  // No operation or process is active
  CmdMessageState.EMPTY               :;
  // Created but not yet started
  CmdMessageState.CREATED             :;
  // Buffered and awaiting execution
  CmdMessageState.BUFFERED            : CommandBuffered    := TRUE;
                                        ParameterAccepted  := TRUE;
  // Buffered in planner for future execution
  CmdMessageState.BUFFERED_IN_PLANNER : CommandBuffered    := TRUE;
                                        ParameterAccepted  := TRUE;
  // Currently active and in progress
  CmdMessageState.ACTIVE              :;
  // Interrupted and awaiting continuation
  CmdMessageState.INTERRUPTED         :;  
  // Requested for abort
  CmdMessageState.ABORT_REQUEST       :;
  // Successfully completed
  CmdMessageState.DONE                : Done               := TRUE;
                                        Busy               := FALSE;
  // Aborted before completion
  CmdMessageState.ABORTED             : Busy               := FALSE;
  // Encountered an error during execution
  CmdMessageState.ERROR               : Error              := TRUE;
                                        Busy               := FALSE;
END_CASE
                
END_METHOD

METHOD INTERNAL ParseResponsePayload : DINT
VAR_INPUT
  /// Response data
  ResponseData : RobotLibraryResponseDataFB;
  /// Timestamp
  Timestamp    : SystemTime;  
END_VAR
VAR
  /// Parameter count
 _parameterCnt : DINT;
END_VAR
// Table 6-445: Received CMD payload (RC to PLC) of "RedefineTrackingPos"
// --------------------------
// Header
// --------------------------
// Byte 00 : USINT      - ParSeq | State     
// Byte 01 : SINT       - AlarmMessageSeverity    
// Byte 02 : UINT       - AlarmMessageCode HB
// Byte 03 :            - AlarmMessageCode LB
// --------------------------
// Datablock
// --------------------------
// Byte 04 : USINT InvocationCounter;
// Byte 05 : SINT  Reserved;
// Byte 06 : INT   OriginID;
// Byte 07 :       OriginID;
                  // call base implementation to parse the header from payload buffer
ResponseData.PayloadPtr := SUPER^.ParseResponsePayload(ResponseData := ResponseData, Timestamp := Timestamp);

// copy parsed header to response
_response.ParSeq                := _rspHeader.ParSeq;
_response.State                 := _rspHeader.State;
_response.AlarmMessageSeverity  := _rspHeader.AlarmMessageSeverity;
_response.AlarmMessageCode      := _rspHeader.AlarmMessageCode;

// Check payload remaining ? 
IF ( ResponseData.IsPayloadRemaining)
THEN 
  // Get Response.InvocationCounter
 _response.InvocationCounter := ResponseData.GetUsint();
  // inc parameter counter
 _parameterCnt := _parameterCnt + 1;
END_IF


// Check payload remaining ? 
IF ( ResponseData.IsPayloadRemaining)
THEN 
  // Get Response.Reserved
  _response.Reserved := ResponseData.GetSint();
  // inc parameter counter
 _parameterCnt := _parameterCnt + 1;
END_IF


// Check payload remaining ? 
IF ( ResponseData.IsPayloadRemaining)
THEN 
  // Get Response.InvocationCounter
 _response.OriginID := ResponseData.GetInt();
  // inc parameter counter
 _parameterCnt := _parameterCnt + 1;
END_IF

 
// Create logging
ParseResponsePayloadLog(ResponseData := ResponseData, Timestamp := Timestamp, ParameterCnt := _parameterCnt);
                
END_METHOD

METHOD INTERNAL ParseResponsePayloadLog
VAR_INPUT
  /// Response data
  ResponseData : RobotLibraryResponseDataFB;
  /// Timestamp
  Timestamp    : SystemTime;  
  /// Parameter count
  ParameterCnt : DINT;
END_VAR
                  // Create log entry for Parameter start
CreateLogMessagePara1 ( Timestamp   := Timestamp,
                        MessageType := MessageType.CMD,
                        Severity    := Severity.DEBUG,
                        MessageCode := 0,
                        MessageText := '{1} parameter(s) to parse from the response data:',
                        Para1       := DINT_TO_STRING(ParameterCnt));
                        

// Return if no parameter is remaining...
IF ( ParameterCnt = 0 ) THEN RETURN; END_IF
// dec remaining parameter(s)                        
ParameterCnt := ParameterCnt - 1;
// Create log entry for InvocationCounter
CreateLogMessagePara1 ( Timestamp   := Timestamp,
                        MessageType := MessageType.CMD,
                        Severity    := Severity.DEBUG,
                        MessageCode := 0,
                        MessageText := 'Response.InvocationCounter = {1}',
                        Para1       :=  USINT_TO_STRING(_response.InvocationCounter));


// Return if no parameter is remaining...
IF ( ParameterCnt = 0 ) THEN RETURN; END_IF
// dec remaining parameter(s)                        
ParameterCnt := ParameterCnt - 1;
// Create log entry for Reserve
CreateLogMessagePara1 ( Timestamp   := Timestamp,
                        MessageType := MessageType.CMD,
                        Severity    := Severity.DEBUG,
                        MessageCode := 0,
                        MessageText := 'Response.Reserve = {1}',
                        Para1       :=  SINT_TO_STRING(_response.Reserved));


// Return if no parameter is remaining...
IF ( ParameterCnt = 0 ) THEN RETURN; END_IF
// dec remaining parameter(s)                        
ParameterCnt := ParameterCnt - 1;
// Create log entry for OriginID
CreateLogMessagePara1 ( Timestamp   := Timestamp,
                        MessageType := MessageType.CMD,
                        Severity    := Severity.DEBUG,
                        MessageCode := 0,
                        MessageText := 'Response.OriginID = {1}',
                        Para1       :=  INT_TO_STRING(_response.OriginID));
                
END_METHOD

METHOD PROTECTED Reset : DINT
VAR_INPUT
END_VAR
                  Reset := SUPER^.Reset();

Done               := FALSE;
Busy               := FALSE;
CommandBuffered    := FALSE;
ParameterAccepted  := FALSE;

                
END_METHOD
END_FUNCTION_BLOCK

/// Synchronize robot with conveyor
FUNCTION_BLOCK MC_SyncToConveyorFB EXTENDS RobotLibraryBaseEnableFB
// ------------------------------------------------------------------------- 
//  SRCI Robot Library                                                
// ------------------------------------------------------------------------- 
//                                                                           
//  Object:      SyncToConveyorFB                                       
//  Author:      Thorsten Brach                                                
//  Date:        2024-06-11
//
//  Description:                                              
//   
//                                                                           
//  Copyright: 
//    (C) 2024 Thorsten Brach. All rights reserved                                                                                                                                            
//             Licensed under the MIT License.
//                                                                           
//  Disclaimer:                                                                           
//    This project is provided without any guarantee and can be used for   
//    private and commercial purposes. Any use is at the user’s 
//    own risk and responsibility.
//
// -------------------------------------------------------------------------
VAR_INPUT
  /// Command parameter 
  ParCmd            : SyncToConveyorParCmd;      
END_VAR

VAR_OUTPUT
  /// Command is transferred and confirmed by the RC
  CommandBuffered   : BOOL;
  /// The command takes control of the motion of the according axis group
  Active            : BOOL;
  /// The command was aborted by another command.
  CommandAborted    : BOOL;
  /// Receiving of input parameter values has been acknowledged by RC
  ParameterAccepted : BOOL;
  /// Command output 
  OutCmd            : SyncToConveyorOutCmd;      
END_VAR

VAR
  /// internal copy of command parameter 
 _parCmd            : SyncToConveyorParCmd;
  /// command data to send
 _command           : SyncToConveyorSendData;
  /// response data received
 _response          : SyncToConveyorRecvData;      
END_VAR

            SUPER^(AxesGroup := AxesGroup);
          

METHOD INTERNAL CheckAddParameter : BOOL
VAR_INPUT
  /// Payload pointer
  PayloadPtr : UDINT;
END_VAR
VAR
  /// Payload as byte array
  Payload    : ARRAY [1..SIZEOF(_command)] OF BYTE;
  /// Null Byte array 
  Null       : ARRAY [1..SIZEOF(_command)] OF BYTE;
  /// Data length to compare
  DataLen    : UDINT;
END_VAR
                  // Payload pointer must be decreased by one byte, because ADR(Payload) is already one byte !
PayloadPtr := LIMIT (0, PayloadPtr - 1, SIZEOF(Payload) -1);
// Convert command struct to payload array
SysDepMemCpy( pDest := ADR(Payload), pSrc := ADR(_command), DataLen := SIZEOF(_command));
// Calculate the data length to compare - at least one byte must be compared !
DataLen := LIMIT(1, SIZEOF(Payload) - PayloadPtr, SIZEOF(Payload)); 
// Compare Payload-Array with Null-Byte-Array
CheckAddParameter := SysDepMemCmp( pData1 := ADR(Payload) + PayloadPtr , pData2 := ADR(Null), DataLen := DataLen) <>  RobotLibraryConstants.OK ;
                
END_METHOD

METHOD PROTECTED CheckFunctionSupported : BOOL
VAR_IN_OUT
  /// Robot assignment of function
  AxesGroup : AxesGroup; 
END_VAR
                  CheckFunctionSupported := AxesGroup.State.RobotData.RCSupportedFunctions.SyncToConveyor;

IF ( NOT CheckFunctionSupported )
THEN
  // call base implementation for set error and create log entry
  SUPER^.CheckFunctionSupported(AxesGroup := AxesGroup);
END_IF
                
END_METHOD

METHOD PROTECTED CheckParameterChanged : BOOL
VAR_IN_OUT
  /// Robot assignment of function
  AxesGroup    : AxesGroup; 
END_VAR
                  // Check ParCmd Size is > 0, because MemCmp does not work correctly with size = 0
IF (SIZEOF(ParCmd) = 0) OR (_stepCmd = 0)
THEN 
  RETURN;
END_IF

// compare memory 
_parameterChanged := ( SysDepMemCmp(pData1 := ADR(ParCmd), pData2 := ADR(_parCmd), DataLen := SIZEOF(ParCmd)) <> RobotLibraryConstants.OK );

// check parameter valid ?
_parameterValid   := CheckParameterValid( AxesGroup := AxesGroup );

IF ((  _parameterChanged        )  AND 
    (  _parameterValid          )) OR
    (  _parameterUpdateInternal )  
THEN  
  // Create log entry for parameter changed event
  CreateLogMessagePara1 ( Timestamp   := AxesGroup.State.SystemTime,
                          MessageType := MessageType.CMD,
                          Severity    := Severity.DEBUG,
                          MessageCode := 0,
                          MessageText := 'NotifyParameterChanged Event {1}',
                          Para1       :=  '' );

  // reset internal flag for send parameter update
 _parameterUpdateInternal := FALSE;
  // update internal copy of parameters 
 _parCmd := ParCmd;
  // inc parameter sequence
 _command.ParSeq := _command.ParSeq + 1;
  // update command data  
  CommandData := CreateCommandPayload(AxesGroup := AxesGroup); // ( Access via reference to rCommandFB in ACR )
  // notify active command register 
  AxesGroup.Acyclic.ActiveCommandRegister.NotifyParameterChanged := _uniqueID;
  // Reset parameter accepted flag
  ParameterAccepted := FALSE;  
END_IF
                
END_METHOD

METHOD PROTECTED CheckParameterValid : BOOL
VAR_IN_OUT
  /// Robot assignment of function
  AxesGroup : AxesGroup; 
END_VAR
                  CheckParameterValid := TRUE;


// Check ParCmd.ConveyorNo valid ? 
IF (( ParCmd.ConveyorNo <   0 ) OR  
    ( ParCmd.ConveyorNo > 255 ))
THEN
  // Parameter not valid
  CheckParameterValid := FALSE;
  // Set error
  SetError( ErrorID := RobotLibraryErrorIdEnum.ERR_INVALID_PAR_CMD, Overwrite := TRUE );
  // Create log entry
  CreateLogMessagePara1 ( Timestamp   := AxesGroup.State.SystemTime,
                          MessageType := MessageType.CMD,
                          Severity    := Severity.ERROR,
                          MessageCode := ErrorID,
                          MessageText := 'Invalid Parameter ParCmd.ConveyorNo = {1}',
                          Para1       :=  USINT_TO_STRING(ParCmd.ConveyorNo));
  RETURN;                          
END_IF


// Check ParCmd.FrameNo valid ? 
IF (( ParCmd.FrameNo <   0                                                 ) OR  
    ( ParCmd.FrameNo > 254                                                 ) OR
    ( ParCmd.FrameNo > AxesGroup.State.ConfigurationData.HighestFrameIndex ) OR
    ( ParCmd.FrameNo > AxesGroup.State.UnifiedFrameIndex                   ))         
THEN
  // Parameter not valid
  CheckParameterValid := FALSE;
  
  // Check FrameNo available on RC ? 
  IF ( ParCmd.FrameNo > AxesGroup.State.ConfigurationData.HighestFrameIndex )
  THEN
    SetError( ErrorID := RobotLibraryErrorIdEnum.ERR_FRAMENO_UNAVAILABLE, Overwrite := TRUE );
  ELSE
    SetError( ErrorID := RobotLibraryErrorIdEnum.ERR_FRAMENO_RANGE, Overwrite := TRUE );
	END_IF  
  
  // Create log entry
  CreateLogMessagePara1 ( Timestamp   := AxesGroup.State.SystemTime,
                          MessageType := MessageType.CMD,
                          Severity    := Severity.ERROR,
                          MessageCode := ErrorID,
                          MessageText := 'Invalid Parameter ParCmd.FrameNo = {1}',
                          Para1       :=  USINT_TO_STRING(ParCmd.FrameNo));
  RETURN;                          
END_IF


// Check ParCmd.SyncInMode valid ? 
IF (( ParCmd.SyncInMode <> SyncInMode.IN_SYNC_IN_ZONE ) AND  
    ( ParCmd.SyncInMode <> SyncInMode.AFTER_DISTANCE  ) AND
    ( ParCmd.SyncInMode <> SyncInMode.AFTER_TIME      ) AND
    ( ParCmd.SyncInMode <> SyncInMode.IMMEDIATELY     ))
THEN
  // Parameter not valid
  CheckParameterValid := FALSE;
  // Set error
  SetError( ErrorID := RobotLibraryErrorIdEnum.ERR_INVALID_PAR_CMD, Overwrite := TRUE );
  // Create log entry
  CreateLogMessagePara1 ( Timestamp   := AxesGroup.State.SystemTime,
                          MessageType := MessageType.CMD,
                          Severity    := Severity.ERROR,
                          MessageCode := ErrorID,
                          MessageText := 'Invalid Parameter ParCmd.SyncInMode = {1}',
                          Para1       :=  SYNC_IN_MODE_TO_STRING(ParCmd.SyncInMode));
  RETURN;                          
END_IF


// Check ParCmd.SyncInParameter valid ? 
IF ( SysDepIsValidReal(ParCmd.SyncInParameter) = FALSE ) 
THEN
  // Parameter not valid
  CheckParameterValid := FALSE;
  // Set error
  SetError( ErrorID := RobotLibraryErrorIdEnum.ERR_INVALID_PAR_CMD, Overwrite := TRUE );
  
  // Create log entry
  CreateLogMessagePara1 ( Timestamp   := AxesGroup.State.SystemTime,
                          MessageType := MessageType.CMD,
                          Severity    := Severity.ERROR,
                          MessageCode := ErrorID,
                          MessageText := 'Invalid Parameter ParCmd.SyncInParameter = {1}',
                          Para1       := VALID_REAL_TO_STRING(ParCmd.SyncInParameter));
  RETURN;                          
END_IF


// Check ParCmd.MaxVelocity valid ? 
IF ( SysDepIsValidReal(ParCmd.MaxVelocity) = FALSE ) 
THEN
  // Parameter not valid
  CheckParameterValid := FALSE;
  // Set error
  SetError( ErrorID := RobotLibraryErrorIdEnum.ERR_INVALID_PAR_CMD, Overwrite := TRUE );
  
  // Create log entry
  CreateLogMessagePara1 ( Timestamp   := AxesGroup.State.SystemTime,
                          MessageType := MessageType.CMD,
                          Severity    := Severity.ERROR,
                          MessageCode := ErrorID,
                          MessageText := 'Invalid Parameter ParCmd.MaxVelocity = {1}',
                          Para1       := VALID_REAL_TO_STRING(ParCmd.MaxVelocity));
  RETURN;                          
END_IF


// Check ParCmd.MaxAcceleration valid ? 
IF ( SysDepIsValidReal(ParCmd.MaxAcceleration) = FALSE ) 
THEN
  // Parameter not valid
  CheckParameterValid := FALSE;
  // Set error
  SetError( ErrorID := RobotLibraryErrorIdEnum.ERR_INVALID_PAR_CMD, Overwrite := TRUE );
  
  // Create log entry
  CreateLogMessagePara1 ( Timestamp   := AxesGroup.State.SystemTime,
                          MessageType := MessageType.CMD,
                          Severity    := Severity.ERROR,
                          MessageCode := ErrorID,
                          MessageText := 'Invalid Parameter ParCmd.MaxAcceleration = {1}',
                          Para1       := VALID_REAL_TO_STRING(ParCmd.MaxAcceleration));
  RETURN;                          
END_IF


// Check ParCmd.ListenerID valid ? 
IF (( ParCmd.ListenerID <   0 ) OR  
    ( ParCmd.ListenerID > 127 ))
THEN
  // Parameter not valid
  CheckParameterValid := FALSE;
  // Set error
  SetError( ErrorID := RobotLibraryErrorIdEnum.ERR_INVALID_PAR_CMD, Overwrite := TRUE );
  // Create log entry
  CreateLogMessagePara1 ( Timestamp   := AxesGroup.State.SystemTime,
                          MessageType := MessageType.CMD,
                          Severity    := Severity.ERROR,
                          MessageCode := ErrorID,
                          MessageText := 'Invalid Parameter ParCmd.ListenerID = {1}',
                          Para1       :=  SINT_TO_STRING(ParCmd.ListenerID));
  RETURN;                          
END_IF
                
END_METHOD

METHOD INTERNAL CreateCommandPayload : RobotLibraryCommandDataFB
VAR_IN_OUT
  /// Robot assignment of function
  AxesGroup : AxesGroup; 
END_VAR
VAR
  /// internal index for loops
 _idx          : DINT;
  /// Parameter count
 _parameterCnt : DINT;
END_VAR
// Table 6-452: Sent CMD payload (PLC to RC) of "SyncToConveyor"
// --------------------------
// Header
// --------------------------
// Byte 00 : UINT       - Type HB     
// Byte 01 :            - Type LB    
// Byte 02 : USINT      - Reserve | ExecutionMode
// Byte 03 : USINT      - ParSeq  | Priority
// --------------------------
// Datablock
// --------------------------
// Byte 04 : SINT       - EmitterID[0]
// Byte 05 : SINT       - EmitterID[1]
// Byte 06 : SINT       - EmitterID[2]
// Byte 07 : SINT       - EmitterID[3]
// Byte 08 : SINT       - ListenerID
// Byte 09 : BYTE       - Reserved
// Byte 10 : USINT      - ConveyorNo
// Byte 11 : USINT      - FrameNo
// Byte 12 : USINT      - SyncInMode
// Byte 13 : REAL       - SyncInParameter HW HB
// Byte 14 :            - SyncInParameter HW LB
// Byte 15 :            - SyncInParameter LW HB
// Byte 16 :            - SyncInParameter LW LB
// Byte 17 : REAL       - MaxVelocity     HW HB
// Byte 18 :            - MaxVelocity     HW LB
// Byte 19 :            - MaxVelocity     LW HB
// Byte 20 :            - MaxVelocity     LW LB
// Byte 21 : REAL       - MaxAcceleration HW HB
// Byte 22 :            - MaxAcceleration HW LB
// Byte 23 :            - MaxAcceleration LW HB
// Byte 24 :            - MaxAcceleration LW LB
// --------------------------
                  // set command parameter 
_command.CmdTyp          :=  CmdType.SyncToConveyor;
_command.ExecMode        :=  ExecMode;
_command.ParSeq          := _command.ParSeq;
_command.Priority        :=  Priority;
_command.EmitterID[0]    := 0;
_command.EmitterID[1]    := 0;
_command.EmitterID[2]    := 0;
_command.EmitterID[3]    := 0;
_command.ListenerID      := _parCmd.ListenerID;
_command.Reserve         := 0;
_command.ConveyorNo      := _parCmd.ConveyorNo;
_command.FrameNo         := _parCmd.FrameNo;
_command.SyncInMode      := _parCmd.SyncInMode;
_command.SyncInParameter := _parCmd.SyncInParameter;
_command.MaxVelocity     := _parCmd.MaxVelocity;
_command.MaxAcceleration := _parCmd.MaxAcceleration;

// copy command data to header
_cmdHeader := _command;
// call base implementation to copy header to payload buffer
CreateCommandPayload := SUPER^.CreateCommandPayload(AxesGroup := AxesGroup);


FOR _idx := 0 TO 3 
DO
  // Check parameter must be added ? 
  IF ( CheckAddParameter(CreateCommandPayload.PayloadPtr))
  THEN
    // add command.EmitterID[x]
    CreateCommandPayload.AddSint(_command.EmitterID[_idx]);
    // inc parameter counter
   _parameterCnt := _parameterCnt + 1;  
  END_IF
END_FOR


// Check parameter must be added ? 
IF ( CheckAddParameter(CreateCommandPayload.PayloadPtr))
THEN
  // add command.ListenerID
  CreateCommandPayload.AddSint(_command.ListenerID);
  // inc parameter counter
 _parameterCnt := _parameterCnt + 1;  
END_IF


// Check parameter must be added ? 
IF ( CheckAddParameter(CreateCommandPayload.PayloadPtr))
THEN
  // add command.Reserve
  CreateCommandPayload.AddByte(_command.Reserve);
  // inc parameter counter
 _parameterCnt := _parameterCnt + 1;  
END_IF


// Check parameter must be added ? 
IF ( CheckAddParameter(CreateCommandPayload.PayloadPtr))
THEN
  // add command.ConveyorNo
  CreateCommandPayload.AddUsint(_command.ConveyorNo);
  // inc parameter counter
 _parameterCnt := _parameterCnt + 1;  
END_IF


// Check parameter must be added ? 
IF ( CheckAddParameter(CreateCommandPayload.PayloadPtr))
THEN
  // add command.FrameNo
  CreateCommandPayload.AddUsint(_command.FrameNo);
  // inc parameter counter
 _parameterCnt := _parameterCnt + 1;  
END_IF


// Check parameter must be added ? 
IF ( CheckAddParameter(CreateCommandPayload.PayloadPtr))
THEN
  // add command.SyncInMode
  CreateCommandPayload.AddUsint(_command.SyncInMode);
  // inc parameter counter
 _parameterCnt := _parameterCnt + 1;  
END_IF


// Check parameter must be added ? 
IF ( CheckAddParameter(CreateCommandPayload.PayloadPtr))
THEN
  // add command.SyncInParameter
  CreateCommandPayload.AddReal(_command.SyncInParameter);
  // inc parameter counter
 _parameterCnt := _parameterCnt + 1;  
END_IF


// Check parameter must be added ? 
IF ( CheckAddParameter(CreateCommandPayload.PayloadPtr))
THEN
  // add command.MaxVelocity
  CreateCommandPayload.AddReal(_command.MaxVelocity);
  // inc parameter counter
 _parameterCnt := _parameterCnt + 1;  
END_IF


// Check parameter must be added ? 
IF ( CheckAddParameter(CreateCommandPayload.PayloadPtr))
THEN
  // add command.MaxAcceleration
  CreateCommandPayload.AddReal(_command.MaxAcceleration);
  // inc parameter counter
 _parameterCnt := _parameterCnt + 1;  
END_IF
  
 
// Create logging
CreateCommandPayloadLog(AxesGroup := AxesGroup, ParameterCnt := _parameterCnt);
                
END_METHOD

METHOD INTERNAL CreateCommandPayloadLog 
VAR_IN_OUT
  /// Robot assignment of function
  AxesGroup : AxesGroup; 
END_VAR
VAR_INPUT
  /// Parameter count
  ParameterCnt : DINT;
END_VAR
VAR 
  /// internal index for loops
 _idx : DINT;
END_VAR
                  // Create log entry for Parameter start
CreateLogMessagePara1 ( Timestamp   := AxesGroup.State.SystemTime,
                        MessageType := MessageType.CMD,
                        Severity    := Severity.DEBUG,
                        MessageCode := 0,
                        MessageText := 'Create command payload with {1} parameter(s) :',
                        Para1       := DINT_TO_STRING(ParameterCnt));

// Create log entry for EmitterID[x]
FOR _idx := 0 TO 3
DO
  // Return if no parameter is remaining...
  IF ( ParameterCnt = 0 ) THEN RETURN; END_IF
  // dec remaining parameter(s)                        
  ParameterCnt := ParameterCnt - 1;
  // Create log entry for Command.EmitterID
  CreateLogMessagePara2 ( Timestamp   := AxesGroup.State.SystemTime,
                          MessageType := MessageType.CMD,
                          Severity    := Severity.DEBUG,
                          MessageCode := 0,
                          MessageText := 'Command.EmitterID[{2}] = {1}',
                          Para1       :=  SINT_TO_STRING(_command.EmitterID[_idx]),
                          Para2       :=  DINT_TO_STRING(_idx));
END_FOR


// Return if no parameter is remaining...
IF ( ParameterCnt = 0 ) THEN RETURN; END_IF
// dec remaining parameter(s)                        
ParameterCnt := ParameterCnt - 1;
// Create log entry for ListenerID
CreateLogMessagePara1 ( Timestamp   := AxesGroup.State.SystemTime,
                        MessageType := MessageType.CMD,
                        Severity    := Severity.DEBUG,
                        MessageCode := 0,
                        MessageText := 'Command.ListenerID = {1}',
                        Para1       :=  SINT_TO_STRING(_command.ListenerID));
                        

// Return if no parameter is remaining...
IF ( ParameterCnt = 0 ) THEN RETURN; END_IF
// dec remaining parameter(s)                        
ParameterCnt := ParameterCnt - 1;
// Create log entry for Reserve
CreateLogMessagePara1 ( Timestamp   := AxesGroup.State.SystemTime,
                        MessageType := MessageType.CMD,
                        Severity    := Severity.DEBUG,
                        MessageCode := 0,
                        MessageText := 'Command.Reserve = {1}',
                        Para1       :=  BYTE_TO_STRING(_command.Reserve));


// Return if no parameter is remaining...
IF ( ParameterCnt = 0 ) THEN RETURN; END_IF
// dec remaining parameter(s)                        
ParameterCnt := ParameterCnt - 1;
// Create log entry for ConveyorNo
CreateLogMessagePara1 ( Timestamp   := AxesGroup.State.SystemTime,
                        MessageType := MessageType.CMD,
                        Severity    := Severity.DEBUG,
                        MessageCode := 0,
                        MessageText := 'Command.ConveyorNo = {1}',
                        Para1       :=  USINT_TO_STRING(_command.ConveyorNo));
                        

// Return if no parameter is remaining...
IF ( ParameterCnt = 0 ) THEN RETURN; END_IF
// dec remaining parameter(s)                        
ParameterCnt := ParameterCnt - 1;
// Create log entry for FrameNo
CreateLogMessagePara1 ( Timestamp   := AxesGroup.State.SystemTime,
                        MessageType := MessageType.CMD,
                        Severity    := Severity.DEBUG,
                        MessageCode := 0,
                        MessageText := 'Command.FrameNo = {1}',
                        Para1       :=  USINT_TO_STRING(_command.FrameNo));       
                        

// Return if no parameter is remaining...
IF ( ParameterCnt = 0 ) THEN RETURN; END_IF
// dec remaining parameter(s)                        
ParameterCnt := ParameterCnt - 1;
// Create log entry for SyncInMode
CreateLogMessagePara1 ( Timestamp   := AxesGroup.State.SystemTime,
                        MessageType := MessageType.CMD,
                        Severity    := Severity.DEBUG,
                        MessageCode := 0,
                        MessageText := 'Command.SyncInMode = {1}',
                        Para1       :=  SYNC_IN_MODE_TO_STRING(_command.SyncInMode));                                         
                        

// Return if no parameter is remaining...
IF ( ParameterCnt = 0 ) THEN RETURN; END_IF
// dec remaining parameter(s)                        
ParameterCnt := ParameterCnt - 1;
// Create log entry for SyncInParameter
CreateLogMessagePara1 ( Timestamp   := AxesGroup.State.SystemTime,
                        MessageType := MessageType.CMD,
                        Severity    := Severity.DEBUG,
                        MessageCode := 0,
                        MessageText := 'Command.SyncInParameter = {1}',
                        Para1       :=  REAL_TO_STRING(_command.SyncInParameter));                                                                 


// Return if no parameter is remaining...
IF ( ParameterCnt = 0 ) THEN RETURN; END_IF
// dec remaining parameter(s)                        
ParameterCnt := ParameterCnt - 1;
// Create log entry for MaxVelocity
CreateLogMessagePara1 ( Timestamp   := AxesGroup.State.SystemTime,
                        MessageType := MessageType.CMD,
                        Severity    := Severity.DEBUG,
                        MessageCode := 0,
                        MessageText := 'Command.MaxVelocity = {1}',
                        Para1       :=  REAL_TO_STRING(_command.MaxVelocity));                                                                 


// Return if no parameter is remaining...
IF ( ParameterCnt = 0 ) THEN RETURN; END_IF
// dec remaining parameter(s)                        
ParameterCnt := ParameterCnt - 1;
// Create log entry for MaxAcceleration
CreateLogMessagePara1 ( Timestamp   := AxesGroup.State.SystemTime,
                        MessageType := MessageType.CMD,
                        Severity    := Severity.DEBUG,
                        MessageCode := 0,
                        MessageText := 'Command.MaxAcceleration = {1}',
                        Para1       :=  REAL_TO_STRING(_command.MaxAcceleration)); 
                
END_METHOD

METHOD FB_init : BOOL
VAR_INPUT
  /// if TRUE, the retain variables are initialized (warm start / cold start)
  bInitRetains : BOOL; 
  /// if TRUE, the instance afterwards gets moved into the copy code (online change)
  bInCopyCode  : BOOL;  
END_VAR
                  MyType := 'MC_SyncToConveyorFB';

ExecMode := ExecutionMode.SEQUENCE_PRIMARY;
Priority := PriorityLevel.NORMAL;
                
END_METHOD

METHOD PROTECTED OnApplyOutCmd
VAR_INPUT
  /// Command message state
  State : CmdMessageState;
END_VAR
                  IF ( State = CmdMessageState.EMPTY ) 
THEN
  // Reset command outputs
  SysDepMemSet(pDest := ADR(OutCmd), Value := 0, DataLen := SIZEOF(OutCmd));         
END_IF

IF ( State = CmdMessageState.ACTIVE )
THEN
  // Update results
  OutCmd.InvocationCounter := _response.InvocationCounter;
  OutCmd.OriginID          := _response.OriginID;
  OutCmd.InSync            := _response.InSync;           
END_IF
                
END_METHOD

METHOD Protected OnExecCancel : DINT
VAR_IN_OUT
  /// Robot assignment of function
  AxesGroup : AxesGroup; 
END_VAR
VAR
  /// internal return value 
 _retVal    : DINT;
END_VAR
                  OnExecCancel := RobotLibraryConstants.RUNNING;

CASE _stepCancel OF
  
  0: // set busy flag
     Busy := TRUE;
    
     // Create log entry
     CreateLogMessagePara1 ( Timestamp   := AxesGroup.State.SystemTime,
                             MessageType := MessageType.CMD,
                             Severity    := Severity.DEBUG,
                             MessageCode := 0,
                             MessageText := 'Execution of {1} cancelled',
                             Para1       := MyType);                 
    
     // try to remove cmd
    _retVal := AxesGroup.Acyclic.ActiveCommandRegister.RemoveCmd(_uniqueID);
  
     // check result of removement       
     IF ( _retVal = RobotLibraryConstants.OK )
     THEN
       // Reset step counter
      _stepCancel := 0;
       // finished okay
       OnExecCancel := RobotLibraryConstants.OK;
     
       // Create log entry
       CreateLogMessagePara1 ( Timestamp   := AxesGroup.State.SystemTime,
                               MessageType := MessageType.CMD,
                               Severity    := Severity.DEBUG,
                               MessageCode := 0,
                               MessageText := '{1} successfully removed from ACR',
                               Para1       := MyType);                 
     ELSE
       // set timeout
       SetTimeout(PT := _timeoutCancel, rTimer := _timerCancel);
       // inc step counter
      _stepCancel := _stepCancel + 1; 
     
       // Create log entry
       CreateLogMessagePara1 ( Timestamp   := AxesGroup.State.SystemTime,
                               MessageType := MessageType.CMD,
                               Severity    := Severity.DEBUG,
                               MessageCode := 0,
                               MessageText := '{1} was not removed from ACR because execution was already in progress',
                               Para1       := MyType);                 
     END_IF       
  
     
 1:  // call clear error 
     OnExecCancel := OnExecErrorClear(AxesGroup := AxesGroup);  
 
     IF ( OnExecCancel = RobotLibraryConstants.OK)
     THEN
       // Reset busy flag
       Busy := FALSE;
       // Reset step counter
      _stepCancel := 0;
       // finished okay
       OnExecCancel := RobotLibraryConstants.OK;
     END_IF  
  
ELSE
  // invalid step
  ErrorID := RobotLibraryErrorIdEnum.ERR_INVALID_STEP;
END_CASE  


                        
// reset step counter
IF (OnExecCancel <> RobotLibraryConstants.RUNNING)
THEN
  // Reset FB variables
  Reset();
  // Reset step counter
 _stepCancel := 0;
END_IF                        
                
END_METHOD

METHOD PROTECTED OnExecErrorClear : DINT
VAR_IN_OUT
  /// Robot assignment of function
  AxesGroup : AxesGroup; 
END_VAR
                  OnExecErrorClear := RobotLibraryConstants.RUNNING;

CASE _stepClearError OF
  
  0:  // set busy flag
      Busy := TRUE;
      // trigger parameter update to disable FB
     _parameterUpdateInternal := TRUE;
      // call Check Parameter changed method to trigger the parameter update to disable the function
      CheckParameterChanged(AxesGroup := AxesGroup);
      // set timeout
      SetTimeout(PT := _timeoutClearError, rTimer := _timerClearError);
      // inc step counter
     _stepClearError := _stepClearError + 1; 
      
  1: IF ( _responseReceived )
     THEN
       // reset response received flag
      _responseReceived := FALSE;
       // reset step counter
      _stepClearError := 0;
       // finished
       OnExecErrorClear := RobotLibraryConstants.OK;
     ELSE
       // timeout exceeded ? 
       IF (CheckTimeout(_timerClearError) = RobotLibraryConstants.OK)
       THEN
         OnExecErrorClear := RobotLibraryConstants.HAS_ERROR;
       END_IF
	   END_IF
ELSE
  // invalid step
  SetError( ErrorID := RobotLibraryErrorIdEnum.ERR_INVALID_STEP, Overwrite := TRUE );
END_CASE


// reset step counter
IF (OnExecErrorClear <> RobotLibraryConstants.RUNNING)
THEN
  // Reset 
  Reset();     
  // reset step counter
 _stepClearError := 0;
END_IF
                
END_METHOD

METHOD PROTECTED OnExecRun : DINT
VAR_IN_OUT
  /// Robot assignment of function
  AxesGroup : AxesGroup; 
END_VAR
                  // call base implementation
SUPER^.OnExecRun(AxesGroup := AxesGroup);

CASE _stepCmd OF
  
  00:  IF ( _enable_R.Q ) AND ( NOT Error) 
       THEN
         // reset the rising edge
        _enable_R();       

         // Check function is supported and parameter are valid ?
         IF (( CheckFunctionSupported( AxesGroup := AxesGroup )) AND
             ( CheckParameterValid   ( AxesGroup := AxesGroup )))      
         THEN
           // Reset all internal flags
           Reset();
           // set busy flag
           Busy := TRUE;
           // Reset command outputs
           SysDepMemSet(pDest := ADR(OutCmd), Value := 0, DataLen := SIZEOF(OutCmd));         
           // apply command parameter
          _parCmd := ParCmd;
           // init parameter sequence
          _command.ParSeq := 1;
           // create command data
           CommandData := CreateCommandPayload(AxesGroup := AxesGroup);
           // Add command to active command register
          _uniqueID := AxesGroup.Acyclic.ActiveCommandRegister.AddCmd( pCommandFB := ADR(THIS^ ));     
           // set timeout
           SetTimeout(PT := _timeoutCmd, rTimer := _timerCmd);
           // inc step counter
          _stepCmd := _stepCmd + 1;
         END_IF 
       END_IF
     

  01:  // Wait for responce received
       IF ( _responseReceived )
       THEN
         // reset response received flag
        _responseReceived := FALSE;
         // update state flags
         OnUpdateStateFlags(_response.State);
         // update state flags
         OnApplyOutCmd(_response.State);
       END_IF

       // do not abort directly, so that the ParSeq update can be send
       IF ( _enable_F.Q ) 
       THEN
         // Set Busy flag
         Busy := TRUE;
         // trigger parameter update to disable FB
        _parameterUpdateInternal := TRUE;
         // reset the falling edge
        _enable_F();
         // set timeout
         SetTimeout(PT := _timeoutCmd, rTimer := _timerCmd);
         // inc step counter
        _stepCmd := _stepCmd + 1; 
       END_IF

      // Wait for response received or timeout or not Initialized
  02: IF ((    _responseReceived                                   )  OR 
          (     CheckTimeout(_timerCmd) = RobotLibraryConstants.OK )) OR 
         (( NOT AxesGroup.State.Initialized                        )  AND
          ( NOT AxesGroup.State.Synchronized                       ))
      THEN
        Reset();   
	    END_IF
      
ELSE
  // invalid step
  SetError( ErrorID := RobotLibraryErrorIdEnum.ERR_INVALID_STEP, Overwrite := TRUE );
END_CASE



// Reset FB
IF (( _enable_R.Q ) OR
    ( _enable_F.Q ))
THEN
  Reset(); 
END_IF
                
END_METHOD

METHOD PROTECTED OnUpdateStateFlags
VAR_INPUT
  /// Command message state
  State : CmdMessageState;
END_VAR
                  // Reset State flags
Active             := FALSE;
CommandAborted     := FALSE;

CASE State OF

  // No operation or process is active
  CmdMessageState.EMPTY               :;
  // Created but not yet started
  CmdMessageState.CREATED             :;
  // Buffered and awaiting execution
  CmdMessageState.BUFFERED            : CommandBuffered    := TRUE;
                                        ParameterAccepted  := TRUE;  
  // Buffered in planner for future execution
  CmdMessageState.BUFFERED_IN_PLANNER : CommandBuffered    := TRUE;
                                        ParameterAccepted  := TRUE;
  // Currently active and in progress
  CmdMessageState.ACTIVE              : Active             := TRUE; 
                                        Enabled            := TRUE;                                        
  // Interrupted and awaiting continuation
  CmdMessageState.INTERRUPTED         :;  
  // Requested for abort
  CmdMessageState.ABORT_REQUEST       :;
  // Successfully completed
  CmdMessageState.DONE                : Busy               := FALSE;
  // Aborted before completion
  CmdMessageState.ABORTED             : CommandAborted     := FALSE;
                                        Busy               := FALSE;
  // Encountered an error during execution
  CmdMessageState.ERROR               : Error              := TRUE;
                                        Busy               := FALSE;
END_CASE
                
END_METHOD

METHOD INTERNAL ParseResponsePayload : DINT
VAR_INPUT
  /// Response data
  ResponseData : RobotLibraryResponseDataFB;
  /// Timestamp
  Timestamp    : SystemTime;  
END_VAR
VAR
  /// Parameter count
 _parameterCnt : DINT;
END_VAR
// Table 6-453: Received CMD payload (RC to PLC) of "SyncToConveyor"
// --------------------------
// Header
// --------------------------
// Byte 00 : USINT      - ParSeq | State     
// Byte 01 : SINT       - AlarmMessageSeverity    
// Byte 02 : UINT       - AlarmMessageCode HB
// Byte 03 :            - AlarmMessageCode LB
// --------------------------
// Datablock
// --------------------------
// Byte 04 : USINT       - InvocationCounter
// Byte 05 : SINT        - Reserved
// Byte 06 : INT         - OriginID
// Byte 07 : BOOL        - InSync
// --------------------------
                  // call base implementation to parse the header from payload buffer
ResponseData.PayloadPtr := SUPER^.ParseResponsePayload(ResponseData := ResponseData, Timestamp := Timestamp);

// copy parsed header to response
_response.ParSeq                := _rspHeader.ParSeq;
_response.State                 := _rspHeader.State;
_response.AlarmMessageSeverity  := _rspHeader.AlarmMessageSeverity;
_response.AlarmMessageCode      := _rspHeader.AlarmMessageCode;


// Check payload remaining ? 
IF ( ResponseData.IsPayloadRemaining)
THEN 
  // Get Response.InvocationCounter
 _response.InvocationCounter := ResponseData.GetUsint();
  // inc parameter counter
 _parameterCnt := _parameterCnt + 1;
END_IF


// Check payload remaining ? 
IF ( ResponseData.IsPayloadRemaining)
THEN 
  // Get Response.Reserved
 _response.Reserved := ResponseData.GetSint();
  // inc parameter counter
 _parameterCnt := _parameterCnt + 1;
END_IF


// Check payload remaining ? 
IF ( ResponseData.IsPayloadRemaining)
THEN 
  // Get Response.InvocationCounter
 _response.OriginID := ResponseData.GetInt();
  // inc parameter counter
 _parameterCnt := _parameterCnt + 1;
END_IF


// Check payload remaining ? 
IF ( ResponseData.IsPayloadRemaining)
THEN 
  // Get Response.InSync
 _response.InSync   := ResponseData.GetBool();
  // inc parameter counter
 _parameterCnt := _parameterCnt + 1;
END_IF


// Create logging
ParseResponsePayloadLog(ResponseData := ResponseData, Timestamp := Timestamp, ParameterCnt := _parameterCnt);
                
END_METHOD

METHOD INTERNAL ParseResponsePayloadLog
VAR_INPUT
  /// Response data
  ResponseData : RobotLibraryResponseDataFB;
  /// Timestamp
  Timestamp    : SystemTime;  
  /// Parameter count
  ParameterCnt : DINT;
END_VAR
                  // Create log entry for Parameter start
CreateLogMessagePara1 ( Timestamp   := Timestamp,
                        MessageType := MessageType.CMD,
                        Severity    := Severity.DEBUG,
                        MessageCode := 0,
                        MessageText := '{1} parameter(s) to parse from the response data:',
                        Para1       := DINT_TO_STRING(ParameterCnt));
                        


// Return if no parameter is remaining...
IF ( ParameterCnt = 0 ) THEN RETURN; END_IF
// dec remaining parameter(s)                        
ParameterCnt := ParameterCnt - 1;
// Create log entry for InvocationCounter
CreateLogMessagePara1 ( Timestamp   := Timestamp,
                        MessageType := MessageType.CMD,
                        Severity    := Severity.DEBUG,
                        MessageCode := 0,
                        MessageText := 'Response.InvocationCounter = {1}',
                        Para1       :=  USINT_TO_STRING(_response.InvocationCounter));


// Return if no parameter is remaining...
IF ( ParameterCnt = 0 ) THEN RETURN; END_IF
// dec remaining parameter(s)                        
ParameterCnt := ParameterCnt - 1;
// Create log entry for Reserve
CreateLogMessagePara1 ( Timestamp   := Timestamp,
                        MessageType := MessageType.CMD,
                        Severity    := Severity.DEBUG,
                        MessageCode := 0,
                        MessageText := 'Response.Reserve = {1}',
                        Para1       :=  SINT_TO_STRING(_response.Reserved));


// Return if no parameter is remaining...
IF ( ParameterCnt = 0 ) THEN RETURN; END_IF
// dec remaining parameter(s)                        
ParameterCnt := ParameterCnt - 1;
// Create log entry for OriginID
CreateLogMessagePara1 ( Timestamp   := Timestamp,
                        MessageType := MessageType.CMD,
                        Severity    := Severity.DEBUG,
                        MessageCode := 0,
                        MessageText := 'Response.OriginID = {1}',
                        Para1       :=  INT_TO_STRING(_response.OriginID));


// Return if no parameter is remaining...
IF ( ParameterCnt = 0 ) THEN RETURN; END_IF
// dec remaining parameter(s)                        
ParameterCnt := ParameterCnt - 1;
// Create log entry for InSync
CreateLogMessagePara1 ( Timestamp   := Timestamp,
                        MessageType := MessageType.CMD,
                        Severity    := Severity.DEBUG,
                        MessageCode := 0,
                        MessageText := 'Response.InSync = {1}',
                        Para1       :=  BOOL_TO_STRING(_response.InSync));
                
END_METHOD

METHOD PROTECTED Reset : DINT
VAR_INPUT
END_VAR
                  SUPER^.Reset();

Busy               := FALSE;
Active             := FALSE;
CommandBuffered    := FALSE;
CommandAborted     := FALSE;
ParameterAccepted  := FALSE;
                
END_METHOD
END_FUNCTION_BLOCK

/// Enables the RC to apply user defined force/ torque through RA’s TCP movement
FUNCTION_BLOCK MC_ForceControlFB EXTENDS RobotLibraryBaseEnableFB
// ------------------------------------------------------------------------- 
//  SRCI Robot Library                                                
// ------------------------------------------------------------------------- 
//                                                                           
//  Object:      ForceControlFB                                       
//  Author:      Thorsten Brach                                                
//  Date:        2024-06-01
//
//  Description:                                              
//   
//                                                                           
//  Copyright: 
//    (C) 2024 Thorsten Brach. All rights reserved                                                                                                                                            
//             Licensed under the MIT License.
//                                                                           
//  Disclaimer:                                                                           
//    This project is provided without any guarantee and can be used for   
//    private and commercial purposes. Any use is at the user’s 
//    own risk and responsibility.
//
// -------------------------------------------------------------------------
VAR_INPUT
  /// Command parameter 
  ParCmd             : ForceControlParCmd;      
END_VAR

VAR_OUTPUT
  /// TRUE, while the following outputs return valid values:
  /// - ForceStatus
  Valid              : BOOL;
  /// Command is transferred and confirmed by the RC
  CommandBuffered    : BOOL;
  /// Receiving of input parameter values has been acknowledged by RC
  ParameterAccepted  : BOOL;
  /// Command output 
  OutCmd             : ForceControlOutCmd;    
END_VAR

VAR
  /// internal copy of command parameter 
 _parCmd            : ForceControlParCmd;
  /// command data to send
 _command           : ForceControlSendData;
  /// response data received
 _response          : ForceControlRecvData;      
END_VAR

            SUPER^(AxesGroup := AxesGroup);
          

METHOD INTERNAL CheckAddParameter : BOOL
VAR_INPUT
  /// Payload pointer
  PayloadPtr : UDINT;
END_VAR
VAR
  /// Payload as byte array
  Payload    : ARRAY [1..SIZEOF(_command)] OF BYTE;
  /// Null Byte array 
  Null       : ARRAY [1..SIZEOF(_command)] OF BYTE;
  /// Data length to compare
  DataLen    : UDINT;
END_VAR
                  // Payload pointer must be decreased by one byte, because ADR(Payload) is already one byte !
PayloadPtr := LIMIT (0, PayloadPtr - 1, SIZEOF(Payload) -1);
// Convert command struct to payload array
SysDepMemCpy( pDest := ADR(Payload), pSrc := ADR(_command), DataLen := SIZEOF(_command));
// Calculate the data length to compare - at least one byte must be compared !
DataLen := LIMIT(1, SIZEOF(Payload) - PayloadPtr, SIZEOF(Payload)); 
// Compare Payload-Array with Null-Byte-Array
CheckAddParameter := SysDepMemCmp( pData1 := ADR(Payload) + PayloadPtr , pData2 := ADR(Null), DataLen := DataLen) <>  RobotLibraryConstants.OK ;
                
END_METHOD

METHOD PROTECTED CheckFunctionSupported : BOOL
VAR_IN_OUT
  /// Robot assignment of function
  AxesGroup : AxesGroup; 
END_VAR
                  CheckFunctionSupported := AxesGroup.State.RobotData.RCSupportedFunctions.ForceControl;

IF ( NOT CheckFunctionSupported )
THEN
  // call base implementation for set error and create log entry
  SUPER^.CheckFunctionSupported(AxesGroup := AxesGroup);
END_IF
                
END_METHOD

METHOD PROTECTED CheckParameterChanged : BOOL
VAR_IN_OUT
  /// Robot assignment of function
  AxesGroup    : AxesGroup; 
END_VAR
                  // Check ParCmd Size is > 0, because MemCmp does not work correctly with size = 0
IF (SIZEOF(ParCmd) = 0) OR (_stepCmd = 0)
THEN 
  RETURN;
END_IF

// compare memory 
_parameterChanged := ( SysDepMemCmp(pData1 := ADR(ParCmd), pData2 := ADR(_parCmd), DataLen := SIZEOF(ParCmd)) <> RobotLibraryConstants.OK );

// check parameter valid ?
_parameterValid   := CheckParameterValid( AxesGroup := AxesGroup );

IF ((  _parameterChanged        )  AND 
    (  _parameterValid          )) OR
    (  _parameterUpdateInternal )  
THEN  
  // Create log entry for parameter changed event
  CreateLogMessagePara1 ( Timestamp   := AxesGroup.State.SystemTime,
                          MessageType := MessageType.CMD,
                          Severity    := Severity.DEBUG,
                          MessageCode := 0,
                          MessageText := 'NotifyParameterChanged Event {1}',
                          Para1       :=  '' );

  // reset internal flag for send parameter update
 _parameterUpdateInternal := FALSE;
  // update internal copy of parameters 
 _parCmd := ParCmd;
  // inc parameter sequence
 _command.ParSeq := _command.ParSeq + 1;
  // update command data  
  CommandData := CreateCommandPayload(AxesGroup := AxesGroup); // ( Access via reference to rCommandFB in ACR )
  // notify active command register 
  AxesGroup.Acyclic.ActiveCommandRegister.NotifyParameterChanged := _uniqueID;
  // Reset Valid output of the FB 
  Valid := FALSE;
  // Reset parameter accepted flag
  ParameterAccepted := FALSE;  
END_IF
                
END_METHOD

METHOD PROTECTED CheckParameterValid : BOOL
VAR_IN_OUT
  /// Robot assignment of function
  AxesGroup : AxesGroup; 
END_VAR
VAR
  /// internal index for loops
 _idx : DINT;
END_VAR
                  CheckParameterValid := TRUE;


// Check ParCmd.ReferenceType valid ? 
IF (( ParCmd.ReferenceType <> ReferenceType.TOOL  ) AND  
    ( ParCmd.ReferenceType <> ReferenceType.FRAME ))
THEN
  // Parameter not valid
  CheckParameterValid := FALSE;
  // Set error
  SetError( ErrorID := RobotLibraryErrorIdEnum.ERR_INVALID_PAR_CMD, Overwrite := TRUE );
  // Create log entry
  CreateLogMessagePara1 ( Timestamp   := AxesGroup.State.SystemTime,
                          MessageType := MessageType.CMD,
                          Severity    := Severity.ERROR,
                          MessageCode := ErrorID,
                          MessageText := 'Invalid Parameter ParCmd.ReferenceType = {1}',
                          Para1       :=  REFERENCE_TYPE_TO_STRING(ParCmd.ReferenceType));
  RETURN;                          
END_IF


FOR _idx := 0 TO 5 
DO
  // Check ParCmd.SensorValue[_idx] valid ? 
  IF ( SysDepIsValidReal(ParCmd.SensorValue[_idx]) = FALSE ) 
  THEN
    // Parameter not valid
    CheckParameterValid := FALSE;
    // Set error
    SetError( ErrorID := RobotLibraryErrorIdEnum.ERR_INVALID_PAR_CMD, Overwrite := TRUE );
    
    // Create log entry
    CreateLogMessagePara2 ( Timestamp   := AxesGroup.State.SystemTime,
                            MessageType := MessageType.CMD,
                            Severity    := Severity.ERROR,
                            MessageCode := ErrorID,
                            MessageText := 'Invalid Parameter ParCmd.SensorValue[{2}] = {1}',
                            Para1       := VALID_REAL_TO_STRING(ParCmd.SensorValue[_idx]),
                            Para2       := DINT_TO_STRING(_idx));
    EXIT;                            
    RETURN;                          
  END_IF
END_FOR


FOR _idx := 0 TO 5 
DO
  // Check ParCmd.TargetValue[_idx] valid ? 
  IF ( SysDepIsValidReal(ParCmd.TargetValue[_idx]) = FALSE ) 
  THEN
    // Parameter not valid
    CheckParameterValid := FALSE;
    // Set error
    SetError( ErrorID := RobotLibraryErrorIdEnum.ERR_INVALID_PAR_CMD, Overwrite := TRUE );
    
    // Create log entry
    CreateLogMessagePara2 ( Timestamp   := AxesGroup.State.SystemTime,
                            MessageType := MessageType.CMD,
                            Severity    := Severity.ERROR,
                            MessageCode := ErrorID,
                            MessageText := 'Invalid Parameter ParCmd.TargetValue[{2}] = {1}',
                            Para1       := VALID_REAL_TO_STRING(ParCmd.TargetValue[_idx]),
                            Para2       := DINT_TO_STRING(_idx));
    EXIT;                            
    RETURN;                          
  END_IF
END_FOR


// Check ParCmd.ToolNo valid ? 
IF (( ParCmd.ToolNo <   0                                                ) OR  
    ( ParCmd.ToolNo > 254                                                ) OR
    ( ParCmd.ToolNo > AxesGroup.State.ConfigurationData.HighestToolIndex ) OR
    ( ParCmd.ToolNo > AxesGroup.State.UnifiedToolIndex                   ))
THEN
  // Parameter not valid
  CheckParameterValid := FALSE;
  
  // Check ToolNo available on RC ? 
  IF ( ParCmd.ToolNo > AxesGroup.State.ConfigurationData.HighestToolIndex )
  THEN
    SetError( ErrorID := RobotLibraryErrorIdEnum.ERR_TOOLNO_UNAVAILABLE, Overwrite := TRUE );
  ELSE
    SetError( ErrorID := RobotLibraryErrorIdEnum.ERR_TOOLNO_RANGE, Overwrite := TRUE );
	END_IF  
  
  // Create log entry
  CreateLogMessagePara1 ( Timestamp   := AxesGroup.State.SystemTime,
                          MessageType := MessageType.CMD,
                          Severity    := Severity.ERROR,
                          MessageCode := ErrorID,
                          MessageText := 'Invalid Parameter ParCmd.ToolNo = {1}',
                          Para1       :=  USINT_TO_STRING(ParCmd.ToolNo));
  RETURN;                          
END_IF


// Check ParCmd.FrameNo valid ? 
IF (( ParCmd.FrameNo <   0                                                 ) OR  
    ( ParCmd.FrameNo > 254                                                 ) OR
    ( ParCmd.FrameNo > AxesGroup.State.ConfigurationData.HighestFrameIndex ) OR
    ( ParCmd.FrameNo > AxesGroup.State.UnifiedFrameIndex                   ))         
THEN
  // Parameter not valid
  CheckParameterValid := FALSE;
  
  // Check FrameNo available on RC ? 
  IF ( ParCmd.FrameNo > AxesGroup.State.ConfigurationData.HighestFrameIndex )
  THEN
    SetError( ErrorID := RobotLibraryErrorIdEnum.ERR_FRAMENO_UNAVAILABLE, Overwrite := TRUE );
  ELSE
    SetError( ErrorID := RobotLibraryErrorIdEnum.ERR_FRAMENO_RANGE, Overwrite := TRUE );
	END_IF  
  
  // Create log entry
  CreateLogMessagePara1 ( Timestamp   := AxesGroup.State.SystemTime,
                          MessageType := MessageType.CMD,
                          Severity    := Severity.ERROR,
                          MessageCode := ErrorID,
                          MessageText := 'Invalid Parameter ParCmd.FrameNo = {1}',
                          Para1       :=  USINT_TO_STRING(ParCmd.FrameNo));
  RETURN;                          
END_IF


// Check ParCmd.ConnectionMode valid ? 
IF (( ParCmd.ConnectionMode <> SensorConnectionMode. RC_SENSOR_ALGORITHM    ) AND  
    ( ParCmd.ConnectionMode <> SensorConnectionMode.PLC_SENSOR_RC_ALGORITHM ) AND
    ( ParCmd.ConnectionMode <> SensorConnectionMode.PLC_SENSOR_RC_ALGORITHM ))
THEN
  // Parameter not valid
  CheckParameterValid := FALSE;
  // Set error
  SetError( ErrorID := RobotLibraryErrorIdEnum.ERR_INVALID_PAR_CMD, Overwrite := TRUE );
  // Create log entry
  CreateLogMessagePara1 ( Timestamp   := AxesGroup.State.SystemTime,
                          MessageType := MessageType.CMD,
                          Severity    := Severity.ERROR,
                          MessageCode := ErrorID,
                          MessageText := 'Invalid Parameter ParCmd.ConnectionMode = {1}',
                          Para1       :=  SENSOR_CONNECTION_MODE_TO_STRING(ParCmd.ConnectionMode));
  RETURN;                          
END_IF


FOR _idx := 0 TO 5 
DO
  // Check ParCmd.SensorFrame[_idx] valid ? 
  IF ( SysDepIsValidReal(ParCmd.SensorFrame[_idx]) = FALSE ) 
  THEN
    // Parameter not valid
    CheckParameterValid := FALSE;
    // Set error
    SetError( ErrorID := RobotLibraryErrorIdEnum.ERR_INVALID_PAR_CMD, Overwrite := TRUE );
    
    // Create log entry
    CreateLogMessagePara2 ( Timestamp   := AxesGroup.State.SystemTime,
                            MessageType := MessageType.CMD,
                            Severity    := Severity.ERROR,
                            MessageCode := ErrorID,
                            MessageText := 'Invalid Parameter ParCmd.SensorFrame[{2}] = {1}',
                            Para1       := VALID_REAL_TO_STRING(ParCmd.SensorFrame[_idx]),
                            Para2       := DINT_TO_STRING(_idx));
    EXIT;                            
    RETURN;                          
  END_IF
END_FOR

// Check ParCmd.CalibrationData valid ? 
IF (( ParCmd.CalibrationData <   0 ) OR  
    ( ParCmd.CalibrationData > 255 ))
THEN
  // Parameter not valid
  CheckParameterValid := FALSE;
  // Set error
  SetError( ErrorID := RobotLibraryErrorIdEnum.ERR_INVALID_PAR_CMD, Overwrite := TRUE );
  // Create log entry
  CreateLogMessagePara1 ( Timestamp   := AxesGroup.State.SystemTime,
                          MessageType := MessageType.CMD,
                          Severity    := Severity.ERROR,
                          MessageCode := ErrorID,
                          MessageText := 'Invalid Parameter ParCmd.CalibrationData = {1}',
                          Para1       :=  USINT_TO_STRING(ParCmd.CalibrationData));
  RETURN;                          
END_IF


// Check ParCmd.TargetWindow valid ? 
IF ( SysDepIsValidReal(ParCmd.TargetWindow) = FALSE ) 
THEN
  // Parameter not valid
  CheckParameterValid := FALSE;
  // Set error
  SetError( ErrorID := RobotLibraryErrorIdEnum.ERR_INVALID_PAR_CMD, Overwrite := TRUE );
  
  // Create log entry
  CreateLogMessagePara1 ( Timestamp   := AxesGroup.State.SystemTime,
                          MessageType := MessageType.CMD,
                          Severity    := Severity.ERROR,
                          MessageCode := ErrorID,
                          MessageText := 'Invalid Parameter ParCmd.TargetWindow = {1}',
                          Para1       := VALID_REAL_TO_STRING(ParCmd.TargetWindow));
  RETURN;                          
END_IF


// Check ParCmd.CompliantAxes valid ? 
IF (( ParCmd.CompliantAxes < 0  ) OR  
    ( ParCmd.CompliantAxes > 63 ))
THEN
  // Parameter not valid
  CheckParameterValid := FALSE;
  // Set error
  SetError( ErrorID := RobotLibraryErrorIdEnum.ERR_INVALID_PAR_CMD, Overwrite := TRUE );
  // Create log entry
  CreateLogMessagePara1 ( Timestamp   := AxesGroup.State.SystemTime,
                          MessageType := MessageType.CMD,
                          Severity    := Severity.ERROR,
                          MessageCode := ErrorID,
                          MessageText := 'Invalid Parameter ParCmd.CompliantAxes = {1}',
                          Para1       :=  BYTE_TO_STRING_BIN(ParCmd.CompliantAxes));
  RETURN;                          
END_IF


// Check ParCmd.MaxVelocity valid ? 
IF ( SysDepIsValidReal(ParCmd.MaxVelocity) = FALSE ) 
THEN
  // Parameter not valid
  CheckParameterValid := FALSE;
  // Set error
  SetError( ErrorID := RobotLibraryErrorIdEnum.ERR_INVALID_PAR_CMD, Overwrite := TRUE );
  
  // Create log entry
  CreateLogMessagePara1 ( Timestamp   := AxesGroup.State.SystemTime,
                          MessageType := MessageType.CMD,
                          Severity    := Severity.ERROR,
                          MessageCode := ErrorID,
                          MessageText := 'Invalid Parameter ParCmd.MaxVelocity = {1}',
                          Para1       := VALID_REAL_TO_STRING(ParCmd.MaxVelocity));
  RETURN;                          
END_IF

FOR _idx := 0 TO 5 
DO
  // Check ParCmd.MaxDeviation[_idx] valid ? 
  IF ( SysDepIsValidReal(ParCmd.MaxDeviation[_idx]) = FALSE ) 
  THEN
    // Parameter not valid
    CheckParameterValid := FALSE;
    // Set error
    SetError( ErrorID := RobotLibraryErrorIdEnum.ERR_INVALID_PAR_CMD, Overwrite := TRUE );
    
    // Create log entry
    CreateLogMessagePara2 ( Timestamp   := AxesGroup.State.SystemTime,
                            MessageType := MessageType.CMD,
                            Severity    := Severity.ERROR,
                            MessageCode := ErrorID,
                            MessageText := 'Invalid Parameter ParCmd.MaxDeviation[{2}] = {1}',
                            Para1       := VALID_REAL_TO_STRING(ParCmd.MaxDeviation[_idx]),
                            Para2       := DINT_TO_STRING(_idx));
    EXIT;                            
    RETURN;                          
  END_IF
END_FOR


// Check ParCmd.ErrorReaction valid ? 
IF (( ParCmd.ErrorReaction <> ErrorReaction.ABORT       ) AND  
    ( ParCmd.ErrorReaction <> ErrorReaction.NO_REACTION ))
THEN
  // Parameter not valid
  CheckParameterValid := FALSE;
  // Set error
  SetError( ErrorID := RobotLibraryErrorIdEnum.ERR_INVALID_PAR_CMD, Overwrite := TRUE );
  // Create log entry
  CreateLogMessagePara1 ( Timestamp   := AxesGroup.State.SystemTime,
                          MessageType := MessageType.CMD,
                          Severity    := Severity.ERROR,
                          MessageCode := ErrorID,
                          MessageText := 'Invalid Parameter ParCmd.ErrorReaction = {1}',
                          Para1       :=  ERROR_REACTION_TO_STRING(ParCmd.ErrorReaction));
  RETURN;                          
END_IF


// Check ParCmd.ErrorReferenceType valid ? 
IF (( ParCmd.ErrorReferenceType <> ReferenceType.TOOL       ) AND  
    ( ParCmd.ErrorReferenceType <> ReferenceType.FRAME ))
THEN
  // Parameter not valid
  CheckParameterValid := FALSE;
  // Set error
  SetError( ErrorID := RobotLibraryErrorIdEnum.ERR_INVALID_PAR_CMD, Overwrite := TRUE );
  // Create log entry
  CreateLogMessagePara1 ( Timestamp   := AxesGroup.State.SystemTime,
                          MessageType := MessageType.CMD,
                          Severity    := Severity.ERROR,
                          MessageCode := ErrorID,
                          MessageText := 'Invalid Parameter ParCmd.ErrorReferenceType = {1}',
                          Para1       :=  REFERENCE_TYPE_TO_STRING(ParCmd.ErrorReferenceType));
  RETURN;                          
END_IF


FOR _idx := 0 TO 5 
DO
  // Check ParCmd.ErrorVector[_idx] valid ? 
  IF ( SysDepIsValidReal(ParCmd.ErrorVector[_idx]) = FALSE ) 
  THEN
    // Parameter not valid
    CheckParameterValid := FALSE;
    // Set error
    SetError( ErrorID := RobotLibraryErrorIdEnum.ERR_INVALID_PAR_CMD, Overwrite := TRUE );
    
    // Create log entry
    CreateLogMessagePara2 ( Timestamp   := AxesGroup.State.SystemTime,
                            MessageType := MessageType.CMD,
                            Severity    := Severity.ERROR,
                            MessageCode := ErrorID,
                            MessageText := 'Invalid Parameter ParCmd.ErrorVector[{2}] = {1}',
                            Para1       := VALID_REAL_TO_STRING(ParCmd.ErrorVector[_idx]),
                            Para2       := DINT_TO_STRING(_idx));
    EXIT;                            
    RETURN;                          
  END_IF
END_FOR


// Check ParCmd.ErrorToolNo valid ? 
IF (( ParCmd.ErrorToolNo < 0   ) OR  
    ( ParCmd.ErrorToolNo > 254 ))
THEN
  // Parameter not valid
  CheckParameterValid := FALSE;
  // Set error
  SetError( ErrorID := RobotLibraryErrorIdEnum.ERR_INVALID_PAR_CMD, Overwrite := TRUE );
  // Create log entry
  CreateLogMessagePara1 ( Timestamp   := AxesGroup.State.SystemTime,
                          MessageType := MessageType.CMD,
                          Severity    := Severity.ERROR,
                          MessageCode := ErrorID,
                          MessageText := 'Invalid Parameter ParCmd.ErrorToolNo = {1}',
                          Para1       :=  USINT_TO_STRING(ParCmd.ErrorToolNo));
  RETURN;                          
END_IF


// Check ParCmd.ErrorFrameNo valid ? 
IF (( ParCmd.ErrorFrameNo < 0   ) OR  
    ( ParCmd.ErrorFrameNo > 254 ))
THEN
  // Parameter not valid
  CheckParameterValid := FALSE;
  // Set error
  SetError( ErrorID := RobotLibraryErrorIdEnum.ERR_INVALID_PAR_CMD, Overwrite := TRUE );
  // Create log entry
  CreateLogMessagePara1 ( Timestamp   := AxesGroup.State.SystemTime,
                          MessageType := MessageType.CMD,
                          Severity    := Severity.ERROR,
                          MessageCode := ErrorID,
                          MessageText := 'Invalid Parameter ParCmd.ErrorFrameNo = {1}',
                          Para1       :=  USINT_TO_STRING(ParCmd.ErrorFrameNo));
  RETURN;                          
END_IF


// Check ParCmd.FixedSensor
// -> no plausibility check for boolean
                
END_METHOD

METHOD INTERNAL CreateCommandPayload : RobotLibraryCommandDataFB
VAR_IN_OUT
  /// Robot assignment of function
  AxesGroup : AxesGroup; 
END_VAR
VAR
  /// Parameter count
 _parameterCnt : DINT;
END_VAR
// Table 6-719: Sent CMD payload (PLC to RC) of "ForceControl"
// --------------------------
// Header
// --------------------------
// Byte 00 : UINT       - Type HB     
// Byte 01 :            - Type LB    
// Byte 02 : USINT      - Reserve | ExecutionMode
// Byte 03 : USINT      - ParSeq  | Priority
// --------------------------
// Datablock
// --------------------------
// Byte 004 : USINT      - ToolNo 
// Byte 005 : USINT      - FrameNo 
// Byte 006 : USINT      - ConnectionMode 
// Byte 007 : BOOL       - FixedSensor
// Byte 008 : REAL       - SensorFrame[0] HW HB
// Byte 009 :            - SensorFrame[0] HW LB
// Byte 010 :            - SensorFrame[0] LW HB
// Byte 011 :            - SensorFrame[0] LW LB
// Byte 012 : REAL       - SensorFrame[1] HW HB
// Byte 013 :            - SensorFrame[1] HW LB
// Byte 014 :            - SensorFrame[1] LW HB
// Byte 015 :            - SensorFrame[1] LW LB
// Byte 016 : REAL       - SensorFrame[2] HW HB
// Byte 017 :            - SensorFrame[2] HW LB
// Byte 018 :            - SensorFrame[2] LW HB
// Byte 019 :            - SensorFrame[2] LW LB
// Byte 020 : REAL       - SensorFrame[3] HW HB
// Byte 021 :            - SensorFrame[3] HW LB
// Byte 022 :            - SensorFrame[3] LW HB
// Byte 023 :            - SensorFrame[3] LW LB
// Byte 024 : REAL       - SensorFrame[4] HW HB
// Byte 025 :            - SensorFrame[4] HW LB
// Byte 026 :            - SensorFrame[4] LW HB
// Byte 027 :            - SensorFrame[4] LW LB
// Byte 028 : REAL       - SensorFrame[5] HW HB
// Byte 029 :            - SensorFrame[5] HW LB
// Byte 030 :            - SensorFrame[5] LW HB
// Byte 031 :            - SensorFrame[5] LW LB
// Byte 032 :            - CalibrationData
// Byte 033 :            - ReferenceType
// Byte 034 : REAL       - SensorValue[0] HW HB
// Byte 035 :            - SensorValue[0] HW LB
// Byte 036 :            - SensorValue[0] LW HB
// Byte 037 :            - SensorValue[0] LW LB
// Byte 038 : REAL       - SensorValue[1] HW HB
// Byte 039 :            - SensorValue[1] HW LB
// Byte 040 :            - SensorValue[1] LW HB
// Byte 041 :            - SensorValue[1] LW LB
// Byte 042 : REAL       - SensorValue[2] HW HB
// Byte 043 :            - SensorValue[2] HW LB
// Byte 044 :            - SensorValue[2] LW HB
// Byte 045 :            - SensorValue[2] LW LB
// Byte 046 : REAL       - SensorValue[3] HW HB
// Byte 047 :            - SensorValue[3] HW LB
// Byte 048 :            - SensorValue[3] LW HB
// Byte 049 :            - SensorValue[3] LW LB
// Byte 050 : REAL       - SensorValue[4] HW HB
// Byte 051 :            - SensorValue[4] HW LB
// Byte 052 :            - SensorValue[4] LW HB
// Byte 053 :            - SensorValue[4] LW LB
// Byte 054 : REAL       - SensorValue[5] HW HB
// Byte 055 :            - SensorValue[5] HW LB
// Byte 056 :            - SensorValue[5] LW HB
// Byte 057 :            - SensorValue[5] LW LB
// Byte 058 : REAL       - SensorValue[5] HW HB
// Byte 059 :            - SensorValue[5] HW LB
// Byte 060 :            - SensorValue[5] LW HB
// Byte 061 :            - SensorValue[5] LW LB
// Byte 062 : REAL       - TargetValue[0] HW HB
// Byte 063 :            - TargetValue[0] HW LB
// Byte 064 :            - TargetValue[0] LW HB
// Byte 065 :            - TargetValue[0] LW LB
// Byte 066 : REAL       - TargetValue[1] HW HB
// Byte 067 :            - TargetValue[1] HW LB
// Byte 068 :            - TargetValue[1] LW HB
// Byte 069 :            - TargetValue[1] LW LB
// Byte 070 : REAL       - TargetValue[2] HW HB
// Byte 071 :            - TargetValue[2] HW LB
// Byte 072 :            - TargetValue[2] LW HB
// Byte 073 :            - TargetValue[2] LW LB
// Byte 074 : REAL       - TargetValue[3] HW HB
// Byte 075 :            - TargetValue[3] HW LB
// Byte 076 :            - TargetValue[3] LW HB
// Byte 077 :            - TargetValue[3] LW LB
// Byte 078 : REAL       - TargetValue[4] HW HB
// Byte 079 :            - TargetValue[4] HW LB
// Byte 080 :            - TargetValue[4] LW HB
// Byte 081 :            - TargetValue[4] LW LB
// Byte 082 : REAL       - TargetValue[5] HW HB
// Byte 083 :            - TargetValue[5] HW LB
// Byte 084 :            - TargetValue[5] LW HB
// Byte 085 :            - TargetValue[5] LW LB
// Byte 086 : UINT       - MaxVelocity LW HB
// Byte 087 :            - MaxVelocity LW LB
// Byte 088 : REAL       - MaxDeviation[0] HW HB
// Byte 089 :            - MaxDeviation[0] HW LB
// Byte 090 :            - MaxDeviation[0] LW HB
// Byte 091 :            - MaxDeviation[0] LW LB
// Byte 092 : REAL       - MaxDeviation[1] HW HB
// Byte 093 :            - MaxDeviation[1] HW LB
// Byte 094 :            - MaxDeviation[1] LW HB
// Byte 095 :            - MaxDeviation[1] LW LB
// Byte 096 : REAL       - MaxDeviation[2] HW HB
// Byte 097 :            - MaxDeviation[2] HW LB
// Byte 098 :            - MaxDeviation[2] LW HB
// Byte 099 :            - MaxDeviation[2] LW LB
// Byte 100 : REAL       - MaxDeviation[3] HW HB
// Byte 101 :            - MaxDeviation[3] HW LB
// Byte 102 :            - MaxDeviation[3] LW HB
// Byte 103 :            - MaxDeviation[3] LW LB
// Byte 104 : REAL       - MaxDeviation[4] HW HB
// Byte 105 :            - MaxDeviation[4] HW LB
// Byte 106 :            - MaxDeviation[4] LW HB
// Byte 107 :            - MaxDeviation[4] LW LB
// Byte 108 : REAL       - MaxDeviation[5] HW HB
// Byte 109 :            - MaxDeviation[5] HW LB
// Byte 110 :            - MaxDeviation[5] LW HB
// Byte 111 :            - MaxDeviation[5] LW LB
// Byte 112 : USINT      - ErrorReaction
// Byte 113 : USINT      - ErrorReferenceType
// Byte 114 : REAL       - ErrorVector[0] HW HB
// Byte 115 :            - ErrorVector[0] HW LB
// Byte 116 :            - ErrorVector[0] LW HB
// Byte 117 :            - ErrorVector[0] LW LB
// Byte 118 : REAL       - ErrorVector[1] HW HB
// Byte 119 :            - ErrorVector[1] HW LB
// Byte 120 :            - ErrorVector[1] LW HB
// Byte 121 :            - ErrorVector[1] LW LB
// Byte 122 : REAL       - ErrorVector[2] HW HB
// Byte 123 :            - ErrorVector[2] HW LB
// Byte 124 :            - ErrorVector[2] LW HB
// Byte 125 :            - ErrorVector[2] LW LB
// Byte 126 : REAL       - ErrorVector[3] HW HB
// Byte 127 :            - ErrorVector[3] HW LB
// Byte 128 :            - ErrorVector[3] LW HB
// Byte 129 :            - ErrorVector[3] LW LB
// Byte 130 : REAL       - ErrorVector[4] HW HB
// Byte 131 :            - ErrorVector[4] HW LB
// Byte 132 :            - ErrorVector[4] LW HB
// Byte 133 :            - ErrorVector[4] LW LB
// Byte 134 : REAL       - ErrorVector[5] HW HB
// Byte 135 :            - ErrorVector[5] HW LB
// Byte 136 :            - ErrorVector[5] LW HB
// Byte 137 :            - ErrorVector[5] LW LB
// Byte 138 : USINT      - ErrorToolNo
// Byte 139 : USINT      - ErrorFrameNo
// Byte 140 : BYTE       - CompliantAxes
// --------------------------
                  // set command parameter 
_command.CmdTyp             :=  CmdType.ForceControl;
_command.ExecMode           :=  ExecMode;
_command.ParSeq             := _command.ParSeq;
_command.Priority           :=  Priority;
_command.ToolNo             := _parCmd.ToolNo;
_command.FrameNo            := _parCmd.FrameNo;
_command.ConnectionMode     := _parCmd.ConnectionMode;
_command.FixedSensor.0      := _parCmd.FixedSensor;
_command.SensorFrame        := _parCmd.SensorFrame;
_command.CalibrationData    := _parCmd.CalibrationData;
_command.ReferenceType      := _parCmd.ReferenceType;
_command.SensorValue        := _parCmd.SensorValue;
_command.TargetValue        := _parCmd.TargetValue;
_command.MaxVelocity        := _parCmd.MaxVelocity;
_command.MaxDeviation       := _parCmd.MaxDeviation;
_command.ErrorReaction      := _parCmd.ErrorReaction;
_command.ErrorReferenceType := _parCmd.ErrorReferenceType;
_command.ErrorVector        := _parCmd.ErrorVector;
_command.ErrorToolNo        := _parCmd.ErrorToolNo;
_command.ErrorFrameNo       := _parCmd.ErrorFrameNo;
_command.CompliantAxes      := _parCmd.CompliantAxes;

// copy command data to header
_cmdHeader := _command;
// call base implementation to copy header to payload buffer
CreateCommandPayload := SUPER^.CreateCommandPayload(AxesGroup := AxesGroup);


// Check parameter must be added ? 
IF ( CheckAddParameter(CreateCommandPayload.PayloadPtr))
THEN
  // add command.ToolNo
  CreateCommandPayload.AddUsint(_command.ToolNo);
  // inc parameter counter
 _parameterCnt := _parameterCnt + 1;  
END_IF


// Check parameter must be added ? 
IF ( CheckAddParameter(CreateCommandPayload.PayloadPtr))
THEN
  // add command.FrameNo
  CreateCommandPayload.AddUsint(_command.FrameNo);
  // inc parameter counter
 _parameterCnt := _parameterCnt + 1;  
END_IF


// Check parameter must be added ? 
IF ( CheckAddParameter(CreateCommandPayload.PayloadPtr))
THEN
  // add command.ConnectionMode
  CreateCommandPayload.AddUsint(_command.ConnectionMode);
  // inc parameter counter
 _parameterCnt := _parameterCnt + 1;  
END_IF


// Check parameter must be added ? 
IF ( CheckAddParameter(CreateCommandPayload.PayloadPtr))
THEN
  // add command.FixedSensor
  CreateCommandPayload.AddByte(_command.FixedSensor);
  // inc parameter counter
 _parameterCnt := _parameterCnt + 1;  
END_IF


// Check parameter must be added ? 
IF ( CheckAddParameter(CreateCommandPayload.PayloadPtr))
THEN
  // add command.SensorFrame[0]
  CreateCommandPayload.AddReal(_command.SensorFrame[0]);
  // inc parameter counter
 _parameterCnt := _parameterCnt + 1;  
END_IF


// Check parameter must be added ? 
IF ( CheckAddParameter(CreateCommandPayload.PayloadPtr))
THEN
  // add command.SensorFrame[1]
  CreateCommandPayload.AddReal(_command.SensorFrame[1]);
  // inc parameter counter
 _parameterCnt := _parameterCnt + 1;  
END_IF


// Check parameter must be added ? 
IF ( CheckAddParameter(CreateCommandPayload.PayloadPtr))
THEN
  // add command.SensorFrame[2]
  CreateCommandPayload.AddReal(_command.SensorFrame[2]);
  // inc parameter counter
 _parameterCnt := _parameterCnt + 1;  
END_IF


// Check parameter must be added ? 
IF ( CheckAddParameter(CreateCommandPayload.PayloadPtr))
THEN
  // add command.SensorFrame[3]
  CreateCommandPayload.AddReal(_command.SensorFrame[3]);
  // inc parameter counter
 _parameterCnt := _parameterCnt + 1;  
END_IF


// Check parameter must be added ? 
IF ( CheckAddParameter(CreateCommandPayload.PayloadPtr))
THEN
  // add command.SensorFrame[4]
  CreateCommandPayload.AddReal(_command.SensorFrame[4]);
  // inc parameter counter
 _parameterCnt := _parameterCnt + 1;  
END_IF


// Check parameter must be added ? 
IF ( CheckAddParameter(CreateCommandPayload.PayloadPtr))
THEN
  // add command.SensorFrame[5]
  CreateCommandPayload.AddReal(_command.SensorFrame[5]);
  // inc parameter counter
 _parameterCnt := _parameterCnt + 1;  
END_IF


// Check parameter must be added ? 
IF ( CheckAddParameter(CreateCommandPayload.PayloadPtr))
THEN
  // add command.CalibrationData
  CreateCommandPayload.AddUsint(_command.CalibrationData);
  // inc parameter counter
 _parameterCnt := _parameterCnt + 1;  
END_IF


// Check parameter must be added ? 
IF ( CheckAddParameter(CreateCommandPayload.PayloadPtr))
THEN
  // add command.CalibrationData
  CreateCommandPayload.AddUInt(_command.ReferenceType);
  // inc parameter counter
 _parameterCnt := _parameterCnt + 1;  
END_IF


// Check parameter must be added ? 
IF ( CheckAddParameter(CreateCommandPayload.PayloadPtr))
THEN
  // add command.SensorValue[0]
  CreateCommandPayload.AddReal(_command.SensorValue[0]);
  // inc parameter counter
 _parameterCnt := _parameterCnt + 1;  
END_IF


// Check parameter must be added ? 
IF ( CheckAddParameter(CreateCommandPayload.PayloadPtr))
THEN
  // add command.SensorValue[1]
  CreateCommandPayload.AddReal(_command.SensorValue[1]);
  // inc parameter counter
 _parameterCnt := _parameterCnt + 1;  
END_IF


// Check parameter must be added ? 
IF ( CheckAddParameter(CreateCommandPayload.PayloadPtr))
THEN
  // add command.SensorValue[2]
  CreateCommandPayload.AddReal(_command.SensorValue[2]);
  // inc parameter counter
 _parameterCnt := _parameterCnt + 1;  
END_IF


// Check parameter must be added ? 
IF ( CheckAddParameter(CreateCommandPayload.PayloadPtr))
THEN
  // add command.SensorValue[3]
  CreateCommandPayload.AddReal(_command.SensorValue[3]);
  // inc parameter counter
 _parameterCnt := _parameterCnt + 1;  
END_IF


// Check parameter must be added ? 
IF ( CheckAddParameter(CreateCommandPayload.PayloadPtr))
THEN
  // add command.SensorValue[4]
  CreateCommandPayload.AddReal(_command.SensorValue[4]);
  // inc parameter counter
 _parameterCnt := _parameterCnt + 1;  
END_IF


// Check parameter must be added ? 
IF ( CheckAddParameter(CreateCommandPayload.PayloadPtr))
THEN
  // add command.SensorValue[5]
  CreateCommandPayload.AddReal(_command.SensorValue[5]);
  // inc parameter counter
 _parameterCnt := _parameterCnt + 1;  
END_IF


// Check parameter must be added ? 
IF ( CheckAddParameter(CreateCommandPayload.PayloadPtr))
THEN
  // add command.TargetValue[0]
  CreateCommandPayload.AddReal(_command.TargetValue[0]);
  // inc parameter counter
 _parameterCnt := _parameterCnt + 1;  
END_IF


// Check parameter must be added ? 
IF ( CheckAddParameter(CreateCommandPayload.PayloadPtr))
THEN
  // add command.TargetValue[1]
  CreateCommandPayload.AddReal(_command.TargetValue[1]);
  // inc parameter counter
 _parameterCnt := _parameterCnt + 1;  
END_IF


// Check parameter must be added ? 
IF ( CheckAddParameter(CreateCommandPayload.PayloadPtr))
THEN
  // add command.TargetValue[2]
  CreateCommandPayload.AddReal(_command.TargetValue[2]);
  // inc parameter counter
 _parameterCnt := _parameterCnt + 1;  
END_IF


// Check parameter must be added ? 
IF ( CheckAddParameter(CreateCommandPayload.PayloadPtr))
THEN
  // add command.TargetValue[3]
  CreateCommandPayload.AddReal(_command.TargetValue[3]);
  // inc parameter counter
 _parameterCnt := _parameterCnt + 1;  
END_IF


// Check parameter must be added ? 
IF ( CheckAddParameter(CreateCommandPayload.PayloadPtr))
THEN
  // add command.TargetValue[4]
  CreateCommandPayload.AddReal(_command.TargetValue[4]);
  // inc parameter counter
 _parameterCnt := _parameterCnt + 1;  
END_IF


// Check parameter must be added ? 
IF ( CheckAddParameter(CreateCommandPayload.PayloadPtr))
THEN
  // add command.TargetValue[5]
  CreateCommandPayload.AddReal(_command.TargetValue[5]);
  // inc parameter counter
 _parameterCnt := _parameterCnt + 1;  
END_IF


// Check parameter must be added ? 
IF ( CheckAddParameter(CreateCommandPayload.PayloadPtr))
THEN
  // add command.MaxVelocity
  CreateCommandPayload.AddUInt(_command.MaxVelocity);
  // inc parameter counter
 _parameterCnt := _parameterCnt + 1;  
END_IF


// Check parameter must be added ? 
IF ( CheckAddParameter(CreateCommandPayload.PayloadPtr))
THEN
  // add command.MaxDeviation[0]
  CreateCommandPayload.AddReal(_command.MaxDeviation[0]);
  // inc parameter counter
 _parameterCnt := _parameterCnt + 1;  
END_IF


// Check parameter must be added ? 
IF ( CheckAddParameter(CreateCommandPayload.PayloadPtr))
THEN
  // add command.MaxDeviation[1]
  CreateCommandPayload.AddReal(_command.MaxDeviation[1]);
  // inc parameter counter
 _parameterCnt := _parameterCnt + 1;  
END_IF


// Check parameter must be added ? 
IF ( CheckAddParameter(CreateCommandPayload.PayloadPtr))
THEN
  // add command.MaxDeviation[2]
  CreateCommandPayload.AddReal(_command.MaxDeviation[2]);
  // inc parameter counter
 _parameterCnt := _parameterCnt + 1;  
END_IF


// Check parameter must be added ? 
IF ( CheckAddParameter(CreateCommandPayload.PayloadPtr))
THEN
  // add command.MaxDeviation[3]
  CreateCommandPayload.AddReal(_command.MaxDeviation[3]);
  // inc parameter counter
 _parameterCnt := _parameterCnt + 1;  
END_IF


// Check parameter must be added ? 
IF ( CheckAddParameter(CreateCommandPayload.PayloadPtr))
THEN
  // add command.MaxDeviation[4]
  CreateCommandPayload.AddReal(_command.MaxDeviation[4]);
  // inc parameter counter
 _parameterCnt := _parameterCnt + 1;  
END_IF


// Check parameter must be added ? 
IF ( CheckAddParameter(CreateCommandPayload.PayloadPtr))
THEN
  // add command.MaxDeviation[5]
  CreateCommandPayload.AddReal(_command.MaxDeviation[5]);
  // inc parameter counter
 _parameterCnt := _parameterCnt + 1;  
END_IF


// Check parameter must be added ? 
IF ( CheckAddParameter(CreateCommandPayload.PayloadPtr))
THEN
  // add command.ErrorReaction
  CreateCommandPayload.AddUsint(_command.ErrorReaction);
  // inc parameter counter
 _parameterCnt := _parameterCnt + 1;  
END_IF


// Check parameter must be added ? 
IF ( CheckAddParameter(CreateCommandPayload.PayloadPtr))
THEN
  // add command.ErrorReferenceType
  CreateCommandPayload.AddUsint(_command.ErrorReferenceType);
  // inc parameter counter
 _parameterCnt := _parameterCnt + 1;  
END_IF


// Check parameter must be added ? 
IF ( CheckAddParameter(CreateCommandPayload.PayloadPtr))
THEN
  // add command.ErrorVector[0]
  CreateCommandPayload.AddReal(_command.ErrorVector[0]);
  // inc parameter counter
 _parameterCnt := _parameterCnt + 1;  
END_IF


// Check parameter must be added ? 
IF ( CheckAddParameter(CreateCommandPayload.PayloadPtr))
THEN
  // add command.ErrorVector[1]
  CreateCommandPayload.AddReal(_command.ErrorVector[1]);
  // inc parameter counter
 _parameterCnt := _parameterCnt + 1;  
END_IF


// Check parameter must be added ? 
IF ( CheckAddParameter(CreateCommandPayload.PayloadPtr))
THEN
  // add command.ErrorVector[2]
  CreateCommandPayload.AddReal(_command.ErrorVector[2]);
  // inc parameter counter
 _parameterCnt := _parameterCnt + 1;  
END_IF


// Check parameter must be added ? 
IF ( CheckAddParameter(CreateCommandPayload.PayloadPtr))
THEN
  // add command.ErrorVector[3]
  CreateCommandPayload.AddReal(_command.ErrorVector[3]);
  // inc parameter counter
 _parameterCnt := _parameterCnt + 1;  
END_IF


// Check parameter must be added ? 
IF ( CheckAddParameter(CreateCommandPayload.PayloadPtr))
THEN
  // add command.ErrorVector[4]
  CreateCommandPayload.AddReal(_command.ErrorVector[4]);
  // inc parameter counter
 _parameterCnt := _parameterCnt + 1;  
END_IF


// Check parameter must be added ? 
IF ( CheckAddParameter(CreateCommandPayload.PayloadPtr))
THEN
  // add command.ErrorVector[5]
  CreateCommandPayload.AddReal(_command.ErrorVector[5]);
  // inc parameter counter
 _parameterCnt := _parameterCnt + 1;  
END_IF


// Check parameter must be added ? 
IF ( CheckAddParameter(CreateCommandPayload.PayloadPtr))
THEN
  // add command.ErrorToolNo
  CreateCommandPayload.AddUsint(_command.ErrorToolNo);
  // inc parameter counter
 _parameterCnt := _parameterCnt + 1;  
END_IF


// Check parameter must be added ? 
IF ( CheckAddParameter(CreateCommandPayload.PayloadPtr))
THEN
  // add command.ErrorFrameNo
  CreateCommandPayload.AddUsint(_command.ErrorFrameNo);
  // inc parameter counter
 _parameterCnt := _parameterCnt + 1;  
END_IF


// Check parameter must be added ? 
IF ( CheckAddParameter(CreateCommandPayload.PayloadPtr))
THEN
  // add command.CompliantAxes
  CreateCommandPayload.AddByte(_command.CompliantAxes);
  // inc parameter counter
 _parameterCnt := _parameterCnt + 1;  
END_IF

  
// Create logging
CreateCommandPayloadLog(AxesGroup := AxesGroup, ParameterCnt := _parameterCnt);
                
END_METHOD

METHOD INTERNAL CreateCommandPayloadLog 
VAR_IN_OUT
  /// Robot assignment of function
  AxesGroup : AxesGroup; 
END_VAR
VAR_INPUT
  /// Parameter count
  ParameterCnt : DINT;
END_VAR
                  // Create log entry for Parameter start
CreateLogMessagePara1 ( Timestamp   := AxesGroup.State.SystemTime,
                        MessageType := MessageType.CMD,
                        Severity    := Severity.DEBUG,
                        MessageCode := 0,
                        MessageText := 'Create command payload with {1} parameter(s) :',
                        Para1       := DINT_TO_STRING(ParameterCnt));


// Return if no parameter is remaining...
IF ( ParameterCnt = 0 ) THEN RETURN; END_IF
// dec remaining parameter(s)                        
ParameterCnt := ParameterCnt - 1;
// Create log entry for ToolNo
CreateLogMessagePara1 ( Timestamp   := AxesGroup.State.SystemTime,
                        MessageType := MessageType.CMD,
                        Severity    := Severity.DEBUG,
                        MessageCode := 0,
                        MessageText := 'Command.ToolNo = {1}',
                        Para1       :=  USINT_TO_STRING(_command.ToolNo));
                        

// Return if no parameter is remaining...
IF ( ParameterCnt = 0 ) THEN RETURN; END_IF
// dec remaining parameter(s)                        
ParameterCnt := ParameterCnt - 1;
// Create log entry for FrameNo
CreateLogMessagePara1 ( Timestamp   := AxesGroup.State.SystemTime,
                        MessageType := MessageType.CMD,
                        Severity    := Severity.DEBUG,
                        MessageCode := 0,
                        MessageText := 'Command.FrameNo = {1}',
                        Para1       :=  USINT_TO_STRING(_command.FrameNo));
                        

// Return if no parameter is remaining...
IF ( ParameterCnt = 0 ) THEN RETURN; END_IF
// dec remaining parameter(s)                        
ParameterCnt := ParameterCnt - 1;
// Create log entry for ConnectionMode
CreateLogMessagePara1 ( Timestamp   := AxesGroup.State.SystemTime,
                        MessageType := MessageType.CMD,
                        Severity    := Severity.DEBUG,
                        MessageCode := 0,
                        MessageText := 'Command.ConnectionMode = {1}',
                        Para1       :=  SENSOR_CONNECTION_MODE_TO_STRING(_command.ConnectionMode));


// Return if no parameter is remaining...
IF ( ParameterCnt = 0 ) THEN RETURN; END_IF
// dec remaining parameter(s)                        
ParameterCnt := ParameterCnt - 1;
// Create log entry for FixedSensor
CreateLogMessagePara1 ( Timestamp   := AxesGroup.State.SystemTime,
                        MessageType := MessageType.CMD,
                        Severity    := Severity.DEBUG,
                        MessageCode := 0,
                        MessageText := 'Command.FixedSensor = {1}',
                        Para1       :=  BYTE_TO_STRING(_command.FixedSensor));


// Return if no parameter is remaining...
IF ( ParameterCnt = 0 ) THEN RETURN; END_IF
// dec remaining parameter(s)                        
ParameterCnt := ParameterCnt - 1;
// Create log entry for SensorFrame[0]
CreateLogMessagePara1 ( Timestamp   := AxesGroup.State.SystemTime,
                        MessageType := MessageType.CMD,
                        Severity    := Severity.DEBUG,
                        MessageCode := 0,
                        MessageText := 'Command.SensorFrame[0] = {1}',
                        Para1       :=  REAL_TO_STRING(_command.SensorFrame[0]));


// Return if no parameter is remaining...
IF ( ParameterCnt = 0 ) THEN RETURN; END_IF
// dec remaining parameter(s)                        
ParameterCnt := ParameterCnt - 1;
// Create log entry for SensorFrame[1]
CreateLogMessagePara1 ( Timestamp   := AxesGroup.State.SystemTime,
                        MessageType := MessageType.CMD,
                        Severity    := Severity.DEBUG,
                        MessageCode := 0,
                        MessageText := 'Command.SensorFrame[1] = {1}',
                        Para1       :=  REAL_TO_STRING(_command.SensorFrame[1]));


// Return if no parameter is remaining...
IF ( ParameterCnt = 0 ) THEN RETURN; END_IF
// dec remaining parameter(s)                        
ParameterCnt := ParameterCnt - 1;
// Create log entry for SensorFrame[2]
CreateLogMessagePara1 ( Timestamp   := AxesGroup.State.SystemTime,
                        MessageType := MessageType.CMD,
                        Severity    := Severity.DEBUG,
                        MessageCode := 0,
                        MessageText := 'Command.SensorFrame[2] = {1}',
                        Para1       :=  REAL_TO_STRING(_command.SensorFrame[2]));


// Return if no parameter is remaining...
IF ( ParameterCnt = 0 ) THEN RETURN; END_IF
// dec remaining parameter(s)                        
ParameterCnt := ParameterCnt - 1;
// Create log entry for SensorFrame[3]
CreateLogMessagePara1 ( Timestamp   := AxesGroup.State.SystemTime,
                        MessageType := MessageType.CMD,
                        Severity    := Severity.DEBUG,
                        MessageCode := 0,
                        MessageText := 'Command.SensorFrame[3] = {1}',
                        Para1       :=  REAL_TO_STRING(_command.SensorFrame[3]));
                                                

// Return if no parameter is remaining...
IF ( ParameterCnt = 0 ) THEN RETURN; END_IF
// dec remaining parameter(s)                        
ParameterCnt := ParameterCnt - 1;
// Create log entry for SensorFrame[4]
CreateLogMessagePara1 ( Timestamp   := AxesGroup.State.SystemTime,
                        MessageType := MessageType.CMD,
                        Severity    := Severity.DEBUG,
                        MessageCode := 0,
                        MessageText := 'Command.SensorFrame[4] = {1}',
                        Para1       :=  REAL_TO_STRING(_command.SensorFrame[4]));
                                                

// Return if no parameter is remaining...
IF ( ParameterCnt = 0 ) THEN RETURN; END_IF
// dec remaining parameter(s)                        
ParameterCnt := ParameterCnt - 1;
// Create log entry for SensorFrame[5]
CreateLogMessagePara1 ( Timestamp   := AxesGroup.State.SystemTime,
                        MessageType := MessageType.CMD,
                        Severity    := Severity.DEBUG,
                        MessageCode := 0,
                        MessageText := 'Command.SensorFrame[5] = {1}',
                        Para1       :=  REAL_TO_STRING(_command.SensorFrame[5]));


// Return if no parameter is remaining...
IF ( ParameterCnt = 0 ) THEN RETURN; END_IF
// dec remaining parameter(s)                        
ParameterCnt := ParameterCnt - 1;
// Create log entry for CalibrationData
CreateLogMessagePara1 ( Timestamp   := AxesGroup.State.SystemTime,
                        MessageType := MessageType.CMD,
                        Severity    := Severity.DEBUG,
                        MessageCode := 0,
                        MessageText := 'Command.CalibrationData = {1}',
                        Para1       :=  USINT_TO_STRING(_command.CalibrationData));
                        

// Return if no parameter is remaining...
IF ( ParameterCnt = 0 ) THEN RETURN; END_IF
// dec remaining parameter(s)                        
ParameterCnt := ParameterCnt - 1;
// Create log entry for ReferenceType
CreateLogMessagePara1 ( Timestamp   := AxesGroup.State.SystemTime,
                        MessageType := MessageType.CMD,
                        Severity    := Severity.DEBUG,
                        MessageCode := 0,
                        MessageText := 'Command.ReferenceType = {1}',
                        Para1       :=  REFERENCE_TYPE_TO_STRING(_command.ReferenceType));                        
                                                

// Return if no parameter is remaining...
IF ( ParameterCnt = 0 ) THEN RETURN; END_IF
// dec remaining parameter(s)                        
ParameterCnt := ParameterCnt - 1;
// Create log entry for SensorValue[0]
CreateLogMessagePara1 ( Timestamp   := AxesGroup.State.SystemTime,
                        MessageType := MessageType.CMD,
                        Severity    := Severity.DEBUG,
                        MessageCode := 0,
                        MessageText := 'Command.SensorValue[0] = {1}',
                        Para1       :=  REAL_TO_STRING(_command.SensorValue[0]));


// Return if no parameter is remaining...
IF ( ParameterCnt = 0 ) THEN RETURN; END_IF
// dec remaining parameter(s)                        
ParameterCnt := ParameterCnt - 1;
// Create log entry for SensorValue[1]
CreateLogMessagePara1 ( Timestamp   := AxesGroup.State.SystemTime,
                        MessageType := MessageType.CMD,
                        Severity    := Severity.DEBUG,
                        MessageCode := 0,
                        MessageText := 'Command.SensorValue[1] = {1}',
                        Para1       :=  REAL_TO_STRING(_command.SensorValue[1]));


// Return if no parameter is remaining...
IF ( ParameterCnt = 0 ) THEN RETURN; END_IF
// dec remaining parameter(s)                        
ParameterCnt := ParameterCnt - 1;
// Create log entry for SensorValue[2]
CreateLogMessagePara1 ( Timestamp   := AxesGroup.State.SystemTime,
                        MessageType := MessageType.CMD,
                        Severity    := Severity.DEBUG,
                        MessageCode := 0,
                        MessageText := 'Command.SensorValue[2] = {1}',
                        Para1       :=  REAL_TO_STRING(_command.SensorValue[2]));


// Return if no parameter is remaining...
IF ( ParameterCnt = 0 ) THEN RETURN; END_IF
// dec remaining parameter(s)                        
ParameterCnt := ParameterCnt - 1;
// Create log entry for SensorValue[3]
CreateLogMessagePara1 ( Timestamp   := AxesGroup.State.SystemTime,
                        MessageType := MessageType.CMD,
                        Severity    := Severity.DEBUG,
                        MessageCode := 0,
                        MessageText := 'Command.SensorValue[3] = {1}',
                        Para1       :=  REAL_TO_STRING(_command.SensorValue[3]));
                                                

// Return if no parameter is remaining...
IF ( ParameterCnt = 0 ) THEN RETURN; END_IF
// dec remaining parameter(s)                        
ParameterCnt := ParameterCnt - 1;
// Create log entry for SensorValue[4]
CreateLogMessagePara1 ( Timestamp   := AxesGroup.State.SystemTime,
                        MessageType := MessageType.CMD,
                        Severity    := Severity.DEBUG,
                        MessageCode := 0,
                        MessageText := 'Command.SensorValue[4] = {1}',
                        Para1       :=  REAL_TO_STRING(_command.SensorValue[4]));
                                                

// Return if no parameter is remaining...
IF ( ParameterCnt = 0 ) THEN RETURN; END_IF
// dec remaining parameter(s)                        
ParameterCnt := ParameterCnt - 1;
// Create log entry for SensorValue[5]
CreateLogMessagePara1 ( Timestamp   := AxesGroup.State.SystemTime,
                        MessageType := MessageType.CMD,
                        Severity    := Severity.DEBUG,
                        MessageCode := 0,
                        MessageText := 'Command.SensorValue[5] = {1}',
                        Para1       :=  REAL_TO_STRING(_command.SensorValue[5]));
                                                

// Return if no parameter is remaining...
IF ( ParameterCnt = 0 ) THEN RETURN; END_IF
// dec remaining parameter(s)                        
ParameterCnt := ParameterCnt - 1;
// Create log entry for TargetValue[0]
CreateLogMessagePara1 ( Timestamp   := AxesGroup.State.SystemTime,
                        MessageType := MessageType.CMD,
                        Severity    := Severity.DEBUG,
                        MessageCode := 0,
                        MessageText := 'Command.TargetValue[0] = {1}',
                        Para1       :=  REAL_TO_STRING(_command.TargetValue[0]));


// Return if no parameter is remaining...
IF ( ParameterCnt = 0 ) THEN RETURN; END_IF
// dec remaining parameter(s)                        
ParameterCnt := ParameterCnt - 1;
// Create log entry for TargetValue[1]
CreateLogMessagePara1 ( Timestamp   := AxesGroup.State.SystemTime,
                        MessageType := MessageType.CMD,
                        Severity    := Severity.DEBUG,
                        MessageCode := 0,
                        MessageText := 'Command.TargetValue[1] = {1}',
                        Para1       :=  REAL_TO_STRING(_command.TargetValue[1]));


// Return if no parameter is remaining...
IF ( ParameterCnt = 0 ) THEN RETURN; END_IF
// dec remaining parameter(s)                        
ParameterCnt := ParameterCnt - 1;
// Create log entry for TargetValue[2]
CreateLogMessagePara1 ( Timestamp   := AxesGroup.State.SystemTime,
                        MessageType := MessageType.CMD,
                        Severity    := Severity.DEBUG,
                        MessageCode := 0,
                        MessageText := 'Command.TargetValue[2] = {1}',
                        Para1       :=  REAL_TO_STRING(_command.TargetValue[2]));


// Return if no parameter is remaining...
IF ( ParameterCnt = 0 ) THEN RETURN; END_IF
// dec remaining parameter(s)                        
ParameterCnt := ParameterCnt - 1;
// Create log entry for TargetValue[3]
CreateLogMessagePara1 ( Timestamp   := AxesGroup.State.SystemTime,
                        MessageType := MessageType.CMD,
                        Severity    := Severity.DEBUG,
                        MessageCode := 0,
                        MessageText := 'Command.TargetValue[3] = {1}',
                        Para1       :=  REAL_TO_STRING(_command.TargetValue[3]));
                                                

// Return if no parameter is remaining...
IF ( ParameterCnt = 0 ) THEN RETURN; END_IF
// dec remaining parameter(s)                        
ParameterCnt := ParameterCnt - 1;
// Create log entry for TargetValue[4]
CreateLogMessagePara1 ( Timestamp   := AxesGroup.State.SystemTime,
                        MessageType := MessageType.CMD,
                        Severity    := Severity.DEBUG,
                        MessageCode := 0,
                        MessageText := 'Command.TargetValue[4] = {1}',
                        Para1       :=  REAL_TO_STRING(_command.TargetValue[4]));
                                                

// Return if no parameter is remaining...
IF ( ParameterCnt = 0 ) THEN RETURN; END_IF
// dec remaining parameter(s)                        
ParameterCnt := ParameterCnt - 1;
// Create log entry for TargetValue[5]
CreateLogMessagePara1 ( Timestamp   := AxesGroup.State.SystemTime,
                        MessageType := MessageType.CMD,
                        Severity    := Severity.DEBUG,
                        MessageCode := 0,
                        MessageText := 'Command.TargetValue[5] = {1}',
                        Para1       :=  REAL_TO_STRING(_command.TargetValue[5]));
                                                

// Return if no parameter is remaining...
IF ( ParameterCnt = 0 ) THEN RETURN; END_IF
// dec remaining parameter(s)                        
ParameterCnt := ParameterCnt - 1;
// Create log entry for MaxVelocity
CreateLogMessagePara1 ( Timestamp   := AxesGroup.State.SystemTime,
                        MessageType := MessageType.CMD,
                        Severity    := Severity.DEBUG,
                        MessageCode := 0,
                        MessageText := 'Command.MaxVelocity = {1}',
                        Para1       :=  UINT_TO_STRING(_command.MaxVelocity));
                        

// Return if no parameter is remaining...
IF ( ParameterCnt = 0 ) THEN RETURN; END_IF
// dec remaining parameter(s)                        
ParameterCnt := ParameterCnt - 1;
// Create log entry for MaxDeviation[0]
CreateLogMessagePara1 ( Timestamp   := AxesGroup.State.SystemTime,
                        MessageType := MessageType.CMD,
                        Severity    := Severity.DEBUG,
                        MessageCode := 0,
                        MessageText := 'Command.MaxDeviation[0] = {1}',
                        Para1       :=  REAL_TO_STRING(_command.MaxDeviation[0]));


// Return if no parameter is remaining...
IF ( ParameterCnt = 0 ) THEN RETURN; END_IF
// dec remaining parameter(s)                        
ParameterCnt := ParameterCnt - 1;
// Create log entry for MaxDeviation[1]
CreateLogMessagePara1 ( Timestamp   := AxesGroup.State.SystemTime,
                        MessageType := MessageType.CMD,
                        Severity    := Severity.DEBUG,
                        MessageCode := 0,
                        MessageText := 'Command.MaxDeviation[1] = {1}',
                        Para1       :=  REAL_TO_STRING(_command.MaxDeviation[1]));


// Return if no parameter is remaining...
IF ( ParameterCnt = 0 ) THEN RETURN; END_IF
// dec remaining parameter(s)                        
ParameterCnt := ParameterCnt - 1;
// Create log entry for MaxDeviation[2]
CreateLogMessagePara1 ( Timestamp   := AxesGroup.State.SystemTime,
                        MessageType := MessageType.CMD,
                        Severity    := Severity.DEBUG,
                        MessageCode := 0,
                        MessageText := 'Command.MaxDeviation[2] = {1}',
                        Para1       :=  REAL_TO_STRING(_command.MaxDeviation[2]));


// Return if no parameter is remaining...
IF ( ParameterCnt = 0 ) THEN RETURN; END_IF
// dec remaining parameter(s)                        
ParameterCnt := ParameterCnt - 1;
// Create log entry for MaxDeviation[3]
CreateLogMessagePara1 ( Timestamp   := AxesGroup.State.SystemTime,
                        MessageType := MessageType.CMD,
                        Severity    := Severity.DEBUG,
                        MessageCode := 0,
                        MessageText := 'Command.MaxDeviation[3] = {1}',
                        Para1       :=  REAL_TO_STRING(_command.MaxDeviation[3]));
                                                

// Return if no parameter is remaining...
IF ( ParameterCnt = 0 ) THEN RETURN; END_IF
// dec remaining parameter(s)                        
ParameterCnt := ParameterCnt - 1;
// Create log entry for MaxDeviation[4]
CreateLogMessagePara1 ( Timestamp   := AxesGroup.State.SystemTime,
                        MessageType := MessageType.CMD,
                        Severity    := Severity.DEBUG,
                        MessageCode := 0,
                        MessageText := 'Command.MaxDeviation[4] = {1}',
                        Para1       :=  REAL_TO_STRING(_command.MaxDeviation[4]));
                                                

// Return if no parameter is remaining...
IF ( ParameterCnt = 0 ) THEN RETURN; END_IF
// dec remaining parameter(s)                        
ParameterCnt := ParameterCnt - 1;
// Create log entry for MaxDeviation[5]
CreateLogMessagePara1 ( Timestamp   := AxesGroup.State.SystemTime,
                        MessageType := MessageType.CMD,
                        Severity    := Severity.DEBUG,
                        MessageCode := 0,
                        MessageText := 'Command.MaxDeviation[5] = {1}',
                        Para1       :=  REAL_TO_STRING(_command.MaxDeviation[5]));                        
                        

// Return if no parameter is remaining...
IF ( ParameterCnt = 0 ) THEN RETURN; END_IF
// dec remaining parameter(s)                        
ParameterCnt := ParameterCnt - 1;
// Create log entry for ErrorReaction
CreateLogMessagePara1 ( Timestamp   := AxesGroup.State.SystemTime,
                        MessageType := MessageType.CMD,
                        Severity    := Severity.DEBUG,
                        MessageCode := 0,
                        MessageText := 'Command.ErrorReaction = {1}',
                        Para1       :=  ERROR_REACTION_TO_STRING(_command.ErrorReaction));    
                        

// Return if no parameter is remaining...
IF ( ParameterCnt = 0 ) THEN RETURN; END_IF
// dec remaining parameter(s)                        
ParameterCnt := ParameterCnt - 1;
// Create log entry for ErrorReferenceType
CreateLogMessagePara1 ( Timestamp   := AxesGroup.State.SystemTime,
                        MessageType := MessageType.CMD,
                        Severity    := Severity.DEBUG,
                        MessageCode := 0,
                        MessageText := 'Command.ErrorReferenceType = {1}',
                        Para1       :=  REFERENCE_TYPE_TO_STRING(_command.ErrorReferenceType));     


// Return if no parameter is remaining...
IF ( ParameterCnt = 0 ) THEN RETURN; END_IF
// dec remaining parameter(s)                        
ParameterCnt := ParameterCnt - 1;
// Create LOG entry FOR ErrorVector[0]
CreateLogMessagePara1 ( Timestamp   := AxesGroup.State.SystemTime,
                        MessageType := MessageType.CMD,
                        Severity    := Severity.DEBUG,
                        MessageCode := 0,
                        MessageText := 'Command.ErrorVector[0] = {1}',
                        Para1       :=  REAL_TO_STRING(_command.ErrorVector[0]));


// Return if no parameter is remaining...
IF ( ParameterCnt = 0 ) THEN RETURN; END_IF
// dec remaining parameter(s)                        
ParameterCnt := ParameterCnt - 1;
// Create log entry for ErrorVector[1]
CreateLogMessagePara1 ( Timestamp   := AxesGroup.State.SystemTime,
                        MessageType := MessageType.CMD,
                        Severity    := Severity.DEBUG,
                        MessageCode := 0,
                        MessageText := 'Command.ErrorVector[1] = {1}',
                        Para1       :=  REAL_TO_STRING(_command.ErrorVector[1]));


// Return if no parameter is remaining...
IF ( ParameterCnt = 0 ) THEN RETURN; END_IF
// dec remaining parameter(s)                        
ParameterCnt := ParameterCnt - 1;
// Create log entry for ErrorVector[2]
CreateLogMessagePara1 ( Timestamp   := AxesGroup.State.SystemTime,
                        MessageType := MessageType.CMD,
                        Severity    := Severity.DEBUG,
                        MessageCode := 0,
                        MessageText := 'Command.ErrorVector[2] = {1}',
                        Para1       :=  REAL_TO_STRING(_command.ErrorVector[2]));


// Return if no parameter is remaining...
IF ( ParameterCnt = 0 ) THEN RETURN; END_IF
// dec remaining parameter(s)                        
ParameterCnt := ParameterCnt - 1;
// Create log entry for ErrorVector[3]
CreateLogMessagePara1 ( Timestamp   := AxesGroup.State.SystemTime,
                        MessageType := MessageType.CMD,
                        Severity    := Severity.DEBUG,
                        MessageCode := 0,
                        MessageText := 'Command.ErrorVector[3] = {1}',
                        Para1       :=  REAL_TO_STRING(_command.ErrorVector[3]));
                                                

// Return if no parameter is remaining...
IF ( ParameterCnt = 0 ) THEN RETURN; END_IF
// dec remaining parameter(s)                        
ParameterCnt := ParameterCnt - 1;
// Create log entry for ErrorVector[4]
CreateLogMessagePara1 ( Timestamp   := AxesGroup.State.SystemTime,
                        MessageType := MessageType.CMD,
                        Severity    := Severity.DEBUG,
                        MessageCode := 0,
                        MessageText := 'Command.ErrorVector[4] = {1}',
                        Para1       :=  REAL_TO_STRING(_command.ErrorVector[4]));
                                                

// Return if no parameter is remaining...
IF ( ParameterCnt = 0 ) THEN RETURN; END_IF
// dec remaining parameter(s)                        
ParameterCnt := ParameterCnt - 1;
// Create log entry for ErrorVector[5]
CreateLogMessagePara1 ( Timestamp   := AxesGroup.State.SystemTime,
                        MessageType := MessageType.CMD,
                        Severity    := Severity.DEBUG,
                        MessageCode := 0,
                        MessageText := 'Command.ErrorVector[5] = {1}',
                        Para1       :=  REAL_TO_STRING(_command.ErrorVector[5]));  


// Return if no parameter is remaining...
IF ( ParameterCnt = 0 ) THEN RETURN; END_IF
// dec remaining parameter(s)                        
ParameterCnt := ParameterCnt - 1;
// Create log entry for ErrorToolNo
CreateLogMessagePara1 ( Timestamp   := AxesGroup.State.SystemTime,
                        MessageType := MessageType.CMD,
                        Severity    := Severity.DEBUG,
                        MessageCode := 0,
                        MessageText := 'Command.ErrorToolNo = {1}',
                        Para1       :=  USINT_TO_STRING(_command.ErrorToolNo));                                                                                        


